0: // Idle
	IF rtWrite.Q AND NOT bBusy THEN
		bBusy 					:= TRUE;
		bError 					:= FALSE;
		udiErrorID				:= 0;
		// MinMon 16#0000_000B;	// 2B
		wSetMinMon.0 			:= bSetMinMon;
		fbADSWRITE.WRITE		:= TRUE;
		fbADSWRITE.IDXOFFS		:= 16#0000_000B;
		fbADSWRITE.LEN			:= 2;
		fbADSWRITE.SRCADDR		:= ADR(wSetMinMon);
		iStepWrite				:= iStepWrite + 5;
	END_IF
	
5, 15, 25: // Wait CMD for end
	fbADSWRITE.WRITE			:= FALSE;
	IF NOT fbADSWRITE.BUSY AND NOT fbADSWRITE.ERR THEN
		iStepWrite				:= iStepWrite + 5;
	ELSIF fbADSWRITE.ERR THEN
		iStepWrite				:= 1000;
	END_IF
	
10: // udiIDXOFFS_MinPos		: UDINT := 16#0000_000D;	// 8B
	fbADSWRITE.WRITE			:= TRUE;
	fbADSWRITE.IDXOFFS			:= 16#0000_000D;
	fbADSWRITE.LEN				:= 8;
	fbADSWRITE.SRCADDR			:= ADR(lrSetMinPos);
	iStepWrite					:= iStepWrite + 5;

20: // 	udiIDXOFFS_MaxMon		: UDINT := 16#0000_000C;	// 2B
	wSetMaxMon.0 				:= bSetMaxMon;
	fbADSWRITE.WRITE			:= TRUE;
	fbADSWRITE.IDXOFFS			:= 16#0000_000C;
	fbADSWRITE.LEN				:= 2;
	fbADSWRITE.SRCADDR			:= ADR(wSetMaxMon);
	iStepWrite					:= iStepWrite + 5;

30: // 		udiIDXOFFS_MaxPos		: UDINT := 16#0000_000E;	// 8B
	fbADSWRITE.WRITE			:= TRUE;
	fbADSWRITE.IDXOFFS			:= 16#0000_000E;
	fbADSWRITE.LEN				:= 8;
	fbADSWRITE.SRCADDR			:= ADR(lrSetMaxPos);
	iStepWrite					:= iStepWrite + 5;
		
35: // 	End
	fbADSWRITE.WRITE			:= FALSE;
	IF NOT fbADSWRITE.BUSY AND NOT fbADSWRITE.ERR THEN
		bBusy 					:= FALSE;
		iStepWrite				:= 0;
	ELSIF fbADSWRITE.ERR THEN
		iStepWrite				:= 1000;
	END_IF
	
1000:
	bBusy 						:= FALSE;
	bError 						:= TRUE;
	udiErrorID					:= fbADSWRITE.ERRID;
	iStepWrite					:= 0;

END_CASE
END_ACTION

END_FUNCTION_BLOCK

// ---- POUs/FB/FB_AxisDiag.TcPOU
//==================================================================================================
//							Beckhoff Automation Poland
//								FB_AxisDiag
//									23.08.2016
//					Blok do diagnostyki osi
// 	v1.0 || TC v 3.1.4020.0 || - pierwsza wersja
//==================================================================================================
FUNCTION_BLOCK FB_AxisDiag
VAR_INPUT
	IPCNetID								: T_AmsNetId; 	(* AmsNetId of the IPC *)
	Timeout								: TIME := DEFAULT_ADS_TIMEOUT;
	Reset								: BOOL;
	GetDiag								: BOOL;
END_VAR
VAR_IN_OUT
	Axis	 								: AXIS_REF;
	stAX5000Diag						: ST_AX5000Diag;
END_VAR
VAR_OUTPUT
	Error								: BOOL;
	AdsErrId							: UINT;
	SercosErrId							: UINT;
	ResetAct							: BOOL;
	DiagAct								: BOOL;
	Busy								: BOOL;
END_VAR
VAR
	iState								: INT;
	iSubState							: INT;
	GetDriveRef							: BOOL := TRUE;
	DriveRef								: ST_DriveRef; (* contains sNetID of EcMaster, nSlaveAddr of EcDrive, nDriveNo of EcDrive, either preset or read from NC *)
	AxisID								: UDINT;

	C1DErrorPrev							: BOOL;
	WcStateErrorPrev						: BOOL;
	AxisErrorPrev							: BOOL;
	OperationalPrev						: BOOL;
	ResetPrev							: BOOL;
	GetDiagPrev							: BOOL;

	fbSoERead							: FB_SoERead;
	fbDiagMessage 						: FB_SoEReadDiagMessage;
	fbClassXDiag							: FB_SoEReadClassXDiag;
	fbDiagNumber						: FB_SoEReadDiagNumber;
	fbDiagNumberList						: FB_SoEReadDiagNumberList;

	fbReset								: FB_SoEReset;
	fbDelay								: TON;
	fbGetSlaveState 						: FB_EcGetSlaveState;
	fbReqSlaveState 						: FB_EcReqSlaveState;
	fbNcReset 							: MC_Reset;

	fbAdsRead							: ADSREAD;
	readBuffer							: ARRAY[0..9] OF BYTE;
	Ids									: T_AmsNetIdArr;

	fbFormatString						: FB_FormatString;
	DiagMsgPrev							: STRING(255);
	LogMsg								: STRING(255);
	strSoEString							: ST_SoE_String;
	I									: INT;
END_VAR
VAR CONSTANT
	NCIDXG_AXPARMS					: UDINT := 16#00004000;	(* Axis with ID: Parameter 			*)
	NCIDXO_AXP_HWAMSADDR			: UDINT := 16#00000031;
END_VAR

stAX5000Diag.bOperational	:= Axis.NcToPlc.StateDWord.0;
stAX5000Diag.bC1DError	 	:= Axis.NcToPlc.StateDWord.28;
stAX5000Diag.bWcStateError 	:= Axis.NcToPlc.StateDWord.30;
stAX5000Diag.bAxisError		:= Axis.NcToPlc.StateDWord.31;
stAX5000Diag.iAxisErrorCode	:= Axis.NcToPlc.ErrorCode;

CASE iState OF
0:	(* idle *)
	GetDriveRef 	:= (DriveRef.nSlaveAddr = 0);

	IF GetDriveRef THEN
		Busy			:= TRUE;
		Error			:= FALSE;
		AdsErrId		:= 0;
		SercosErrId		:= 0;
		iState 			:= 1;
		iSubState		:= 0;
		AxisID 			:= Axis.NcToPlc.AxisId;

	ELSIF Reset AND NOT ResetPrev THEN
		Busy			:= TRUE;
		ResetAct		:= TRUE;
		ResetPrev		:= Reset;
		Error			:= FALSE;
		AdsErrId		:= 0;
		SercosErrId		:= 0;
		iState 			:= 2;
		iSubState		:= 0;
		AxisID 			:= Axis.NcToPlc.AxisId;

	ELSIF GetDiag AND NOT GetDiagPrev OR
		(stAX5000Diag.bC1DError AND NOT C1DErrorPrev) OR (NOT stAX5000Diag.bC1DError AND C1DErrorPrev) (* rising/falling C1D *) OR
		(stAX5000Diag.bWcStateError AND NOT WcStateErrorPrev) OR (NOT stAX5000Diag.bWcStateError AND WcStateErrorPrev) (* rising/falling WcState *) OR
		(stAX5000Diag.bAxisError AND NOT AxisErrorPrev) OR (NOT stAX5000Diag.bAxisError AND AxisErrorPrev) (* rising/falling NcError *) OR
		(stAX5000Diag.bOperational AND NOT OperationalPrev) OR (NOT stAX5000Diag.bOperational AND OperationalPrev) (* rising/falling Enable *) THEN

		Busy			:= TRUE;
		DiagAct			:= TRUE;
		GetDiagPrev		:= GetDiag;
		Error			:= FALSE;
		AdsErrId		:= 0;
		SercosErrId		:= 0;
		iState 			:= 3;
		iSubState		:= 0;
		AxisID 			:= Axis.NcToPlc.AxisId;

		(* set/clear flags *)
		C1DErrorPrev		:= stAX5000Diag.bC1DError;
		WcStateErrorPrev	:= stAX5000Diag.bWcStateError;
		AxisErrorPrev		:= stAX5000Diag.bAxisError;
		OperationalPrev		:= stAX5000Diag.bOperational;

	ELSE
		ResetAct	:= FALSE;
		DiagAct		:= FALSE;
	END_IF

1:	(* get drive reference *)
	M_GetDriveRef();

2:	(* reset and state change *)
	M_Reset();

3:	(* get diag data *)
	M_GetDiagnosis();

END_CASE

(* clear latch *)
ResetPrev	:= ResetPrev AND Reset;
GetDiagPrev	:= GetDiagPrev AND GetDiag;

ACTION M_GetDiagnosis:
CASE iSubState OF
0:	fbClassXDiag(
		NetId		:= IPCNetID,
		Execute		:= TRUE,
		DiagClass 	:= 1,
		Timeout		:= DEFAULT_ADS_TIMEOUT,
		Axis		:= Axis,
	);

	IF NOT fbClassXDiag.Busy THEN
		fbClassXDiag(Execute:= FALSE,Axis := Axis);

		IF NOT fbClassXDiag.Error THEN
			stAX5000Diag.wClass1Diag	:= fbClassXDiag.ClassXDiag;
			stAX5000Diag.stClass1Diag	:= F_ConvWordToSTAX5000C1D(stAX5000Diag.wClass1Diag);
		ELSE
			Error			:= TRUE;
			AdsErrId		:= fbClassXDiag.AdsErrId;
			SercosErrId	:= fbClassXDiag.SercosErrId;
		END_IF
		iSubState	:= iSubState + 1;
	END_IF

1:	fbDiagMessage(
		NetId	:= IPCNetID,
		Execute	:= TRUE,
		Timeout	:= DEFAULT_ADS_TIMEOUT,
		Axis	:= Axis,
	);

	IF NOT fbDiagMessage.Busy THEN
		fbDiagMessage(Execute:= FALSE,Axis := Axis);

		IF NOT fbDiagMessage.Error THEN
			stAX5000Diag.strDiagMessage := LEFT(fbDiagMessage.DiagMessage.strData, UINT_TO_INT(fbDiagMessage.DiagMessage.iActualSize));
		ELSE
			Error			:= TRUE;
			AdsErrId		:= fbDiagMessage.AdsErrId;
			SercosErrId	:= fbDiagMessage.SercosErrId;
		END_IF
		iSubState	:= iSubState + 1;
	END_IF

2:	fbDiagNumber(
		NetId	:= IPCNetID,
		Execute	:= TRUE,
		Timeout	:= DEFAULT_ADS_TIMEOUT,
		Axis	:= Axis,
	);

	IF NOT fbDiagNumber.Busy THEN
		fbDiagNumber(Execute:= FALSE,Axis := Axis);

		IF NOT fbDiagNumber.Error THEN
			stAX5000Diag.iDiagNumber := fbDiagNumber.DiagNumber;
		ELSE
			Error			:= TRUE;
			AdsErrId		:= fbDiagNumber.AdsErrId;
			SercosErrId	:= fbDiagNumber.SercosErrId;
		END_IF
		iSubState	:= iSubState + 1;
	END_IF

3:	fbSoERead(
		NetId	:= IPCNetID,
		Execute	:= TRUE,
		Idn		:= 135,
		Element	:=16#44,
		pDstBuf	:=ADR(stAX5000Diag.wDriveStatus),
		BufLen	:=SIZEOF(stAX5000Diag.wDriveStatus),
		Timeout	:= DEFAULT_ADS_TIMEOUT,
		Axis	:= Axis,
	);

	IF NOT fbSoERead.Busy THEN
		fbSoERead(Execute:= FALSE,Axis := Axis);
		IF NOT fbSoERead.Error THEN
			stAX5000Diag.stDriveStatus := F_ConvWordToSTAX5000DriveStatus(stAX5000Diag.wDriveStatus);
			iSubState		:= iSubState + 1;
		ELSE
			Error			:= TRUE;
			AdsErrId		:= fbSoERead.AdsErrId;
			SercosErrId	:= fbSoERead.SercosErrId;
			iSubState		:= iSubState + 2;
		END_IF
	END_IF

4:	fbSoERead(
		NetId	:= IPCNetID,
		Execute	:= TRUE,
		Idn		:= stAX5000Diag.stDriveStatus.iActOpModeParNum,
		Element	:=16#44,
		pDstBuf	:=ADR(stAX5000Diag.stDriveStatus.eActOpMode),
		BufLen	:=SIZEOF(stAX5000Diag.stDriveStatus.eActOpMode),
		Timeout	:= DEFAULT_ADS_TIMEOUT,
		Axis	:= Axis,
	);

	IF NOT fbSoERead.Busy THEN
		fbSoERead(Execute:= FALSE,Axis := Axis);
		IF NOT fbSoERead.Error THEN
			;
		ELSE
			Error			:= TRUE;
			AdsErrId		:= fbSoERead.AdsErrId;
			SercosErrId	:= fbSoERead.SercosErrId;
		END_IF
		iSubState	:= iSubState + 1;
	END_IF

5:	fbGetSlaveState(
		sNetId		:= DriveRef.sNetId,
		nSlaveAddr	:= DriveRef.nSlaveAddr,
		bExecute	:= TRUE,
		tTimeout	:= DEFAULT_ADS_TIMEOUT,
	);

	IF NOT fbGetSlaveState.bBusy THEN
		fbGetSlaveState(bExecute:= FALSE);
		IF NOT fbGetSlaveState.bError THEN
			stAX5000Diag.stEcSlaveState := fbGetSlaveState.state;
			stAX5000Diag.stEcSlaveStateBits := F_ConvSlaveStateToBits(fbGetSlaveState.state);
		ELSE
			Error			:= TRUE;
			AdsErrId		:= UDINT_TO_UINT(fbGetSlaveState.nErrId);
		END_IF

		IF stAX5000Diag.stEcSlaveStateBits.bError THEN
			IF stAX5000Diag.stEcSlaveStateBits.bPreop THEN
				(* read S21 - IDN List of Invalid operation data for CP2 (Preop->SaveOp) *)
				MEMSET(ADR(stAX5000Diag.stCPxInvParamList), 0, SIZEOF(stAX5000Diag.stCPxInvParamList));
				stAX5000Diag.bPreopToSafeOpError := TRUE;
				stAX5000Diag.bSafeOpToOpError := FALSE;
				iSubState	:= iSubState + 1;
			ELSIF stAX5000Diag.stEcSlaveStateBits.bSafeOp THEN
				(* read S22 - IDN List of Invalid operation data for CP3 (SaveOp->Op) *)
				MEMSET(ADR(stAX5000Diag.stCPxInvParamList), 0, SIZEOF(stAX5000Diag.stCPxInvParamList));
				stAX5000Diag.bPreopToSafeOpError := FALSE;
				stAX5000Diag.bSafeOpToOpError := TRUE;
				iSubState	:= iSubState + 2;
			ELSE
				(* Skip S21 + S22 *)
				MEMSET(ADR(stAX5000Diag.stCPxInvParamList), 0, SIZEOF(stAX5000Diag.stCPxInvParamList));
				stAX5000Diag.bPreopToSafeOpError := FALSE;
				stAX5000Diag.bSafeOpToOpError := FALSE;
				iSubState	:= iSubState + 3;
			END_IF
		ELSE
			(* Skip S21 + S22 *)
			MEMSET(ADR(stAX5000Diag.stCPxInvParamList), 0, SIZEOF(stAX5000Diag.stCPxInvParamList));
			stAX5000Diag.bPreopToSafeOpError := FALSE;
			stAX5000Diag.bSafeOpToOpError := FALSE;
			iSubState	:= iSubState + 3;
		END_IF
	END_IF

6:	(* read S21 - IDN List of Invalid operation data for CP2 (Preop->SaveOp) *)
	fbSoERead(
		NetId	:= IPCNetID,
		Execute	:= TRUE,
		Idn		:= 21,
		Element	:=16#40,
		pDstBuf	:=ADR(stAX5000Diag.stCPxInvParamList),
		BufLen	:=SIZEOF(stAX5000Diag.stCPxInvParamList),
		Timeout	:= DEFAULT_ADS_TIMEOUT,
		Axis	:= Axis,
	);

	IF NOT fbSoERead.Busy THEN
		fbSoERead(Execute:= FALSE,Axis := Axis);
		IF NOT fbSoERead.Error THEN
			;
		ELSE
			Error			:= TRUE;
			AdsErrId		:= fbSoERead.AdsErrId;
			SercosErrId	:= fbSoERead.SercosErrId;
		END_IF
		iSubState	:= iSubState + 2;
	END_IF

7:	(* read S22 - IDN List of Invalid operation data for CP3 (SaveOp->Op) *)
	fbSoERead(
		NetId	:= IPCNetID,
		Execute	:= TRUE,
		Idn		:= 22,
		Element	:=16#40,
		pDstBuf	:=ADR(stAX5000Diag.stCPxInvParamList),
		BufLen	:=SIZEOF(stAX5000Diag.stCPxInvParamList),
		Timeout	:= DEFAULT_ADS_TIMEOUT,
		Axis	:= Axis,
	);

	IF NOT fbSoERead.Busy THEN
		fbSoERead(Execute:= FALSE,Axis := Axis);
		IF NOT fbSoERead.Error THEN
			;
		ELSE
			Error			:= TRUE;
			AdsErrId		:= fbSoERead.AdsErrId;
			SercosErrId	:= fbSoERead.SercosErrId;
		END_IF
		iSubState	:= iSubState + 1;
	END_IF

8:	fbDiagNumberList(
		NetId			:= IPCNetID,
		Execute			:= TRUE,
		Timeout			:= DEFAULT_ADS_TIMEOUT,
		pDiagNumber		:= ADR(stAX5000Diag.stDiagNumberList),
		Size			:= SIZEOF(stAX5000Diag.stDiagNumberList),
		Axis			:= Axis,
	);

	IF NOT fbDiagNumberList.Busy THEN
		fbDiagNumberList(Execute:= FALSE,Axis := Axis);

		IF NOT fbDiagNumberList.Error THEN
			IF GVL_AXIS.bLogDriveDiagMsgs THEN
				IF (stAX5000Diag.strDiagMessage <> DiagMsgPrev) AND (stAX5000Diag.stDiagNumberList.iActualSize > 0) THEN

					fbFormatString(
						sFormat := 'Axis ID: %d, DriveDiag: ',
						arg1 := F_UDINT(AxisID),
						sOut => LogMsg
					);
	
					FOR I := 0 TO MIN(29, UINT_TO_INT(stAX5000Diag.stDiagNumberList.iActualSize)/4-1) DO
						IF (stAX5000Diag.stDiagNumberList.arrDiagNumbers[I] <> 0) THEN
							fbFormatString(
								sFormat := '%X, ',
								arg1 := F_UDINT(stAX5000Diag.stDiagNumberList.arrDiagNumbers[I])
							);
	
							LogMsg := CONCAT(LogMsg, fbFormatString.sOut);
						END_IF
					END_FOR
	
					LogMsg := CONCAT(LogMsg, 'DiagMsg: ');
					LogMsg := CONCAT(LogMsg, stAX5000Diag.strDiagMessage);
	
					(* report message *)
					ADSLOGSTR(msgCtrlMask := ADSLOG_MSGTYPE_ERROR OR ADSLOG_MSGTYPE_LOG,
						msgFmtStr := LogMsg, strArg:= '');
	
					DiagMsgPrev := stAX5000Diag.strDiagMessage;
				END_IF
			END_IF
		ELSE
			Error			:= TRUE;
			AdsErrId		:= fbDiagNumberList.AdsErrId;
			SercosErrId	:= fbDiagNumberList.SercosErrId;
		END_IF

		IF (stAX5000Diag.strMotorType = '') OR (stAX5000Diag.strDriveType = '') THEN
			iSubState	:= iSubState + 1;
		ELSE
			DiagAct	:= FALSE;
			iSubState	:= 0;
			iState		:= 0;
			Busy		:= FALSE;
		END_IF
	END_IF

9:	fbSoERead(
		NetId	:= IPCNetID,
		Execute	:= TRUE,
		Idn		:= P_0_IDN + 53,
		Element	:=16#44,
		pDstBuf	:=ADR(strSoEString),
		BufLen	:=SIZEOF(strSoEString),
		Timeout	:= DEFAULT_ADS_TIMEOUT,
		Axis	:= Axis,
	);

	IF NOT fbSoERead.Busy THEN
		fbSoERead(Execute:= FALSE,Axis := Axis);
		IF NOT fbSoERead.Error THEN
			MEMSET(ADR(stAX5000Diag.strMotorType),0,SIZEOF(stAX5000Diag.strMotorType));
			MEMCPY(ADR(stAX5000Diag.strMotorType),ADR(strSoEString.strData),MIN(SIZEOF(stAX5000Diag.strMotorType),strSoEString.iActualSize));
		ELSE
			Error			:= TRUE;
			AdsErrId		:= fbSoERead.AdsErrId;
			SercosErrId	:= fbSoERead.SercosErrId;
		END_IF
		iSubState	:= iSubState + 1;
	END_IF

10:	fbSoERead(
		NetId	:= IPCNetID,
		Execute	:= TRUE,
		Idn		:= P_0_IDN + 324,
		Element	:=16#44,
		pDstBuf	:=ADR(strSoEString),
		BufLen	:=SIZEOF(strSoEString),
		Timeout	:= DEFAULT_ADS_TIMEOUT,
		Axis	:= Axis,
	);

	IF NOT fbSoERead.Busy THEN
		fbSoERead(Execute:= FALSE,Axis := Axis);
		IF NOT fbSoERead.Error THEN
			MEMSET(ADR(stAX5000Diag.strDriveType),0,SIZEOF(stAX5000Diag.strDriveType));
			MEMCPY(ADR(stAX5000Diag.strDriveType),ADR(strSoEString.strData),MIN(SIZEOF(stAX5000Diag.strDriveType),strSoEString.iActualSize));
		ELSE
			Error			:= TRUE;
			AdsErrId		:= fbSoERead.AdsErrId;
			SercosErrId	:= fbSoERead.SercosErrId;
		END_IF
		DiagAct	:= FALSE;
		iSubState	:= 0;
		iState		:= 0;
		Busy		:= FALSE;
	END_IF


END_CASE
END_ACTION

ACTION M_GetDriveRef:
(* get reference from NC *)
fbAdsRead(
	NETID	:= IPCNetID,
	PORT	:= AMSPORT_R0_NC,
	IDXGRP	:= NCIDXG_AXPARMS + Axis.NcToPlc.AxisId,
	IDXOFFS	:= NCIDXO_AXP_HWAMSADDR,
	LEN		:= SIZEOF(readBuffer) ,
	DESTADDR:= ADR(readBuffer),
	READ	:= TRUE,
	TMOUT	:= Timeout
);

IF NOT fbAdsRead.BUSY THEN
	fbAdsRead(READ := FALSE);
	stAX5000Diag.nNCAxisID := Axis.NcToPlc.AxisId;

	IF NOT fbAdsRead.ERR THEN
		MEMCPY(ADR(Ids), ADR(readBuffer), SIZEOF(Ids)); 										(* readBuffer[0..5] *)
		MEMCPY(ADR(DriveRef.nSlaveAddr), ADR(readBuffer[6]), SIZEOF(DriveRef.nSlaveAddr));  	(* readBuffer[6..7] *)
		MEMCPY(ADR(DriveRef.nDriveNo), ADR(readBuffer[8]), SIZEOF(DriveRef.nDriveNo));  		(* readBuffer[8..9] *)

		(* create string out of byte array *)
		DriveRef.sNetId := F_CreateAmsNetId(Ids);
		GetDriveRef := FALSE;
	END_IF

	Busy	:= FALSE;
	iState	:= 0;
END_IF
END_ACTION

ACTION M_Reset:
CASE iSubState OF
0:
	IF stAX5000Diag.bWcStateError OR stAX5000Diag.bC1DError THEN
		(* ResetAmplifier *)
		iSubState := iSubState + 1;
	ELSIF stAX5000Diag.stEcSlaveStateBits.bError AND GVL_Axis.bForceStateChgAfterDrvReset THEN
		(* Clear Error *)
		iSubState := 4;
	ELSIF (NOT stAX5000Diag.bOperational) OR stAX5000Diag.bAxisError OR (stAX5000Diag.iAxisErrorCode <> 0) THEN
		(* NC Reset only *)
		iSubState := 6;
	ELSE
		(* reset not required *)
		iSubState	:= 0;
		iState		:= 0;
		Busy		:= FALSE;
		ResetAct	:= FALSE;
	END_IF

1:	(* ResetAmplifier *)
	fbReset(
		NetId	:= IPCNetID,
		Execute	:= TRUE,
		Timeout	:= DEFAULT_ADS_TIMEOUT,
		Axis	:= Axis,
	);
	IF NOT fbReset.Busy THEN
		fbReset(Execute:= FALSE, Axis:= Axis);

		IF NOT fbReset.Error THEN
			IF GVL_Axis.bLogDriveDiagMsgs THEN
				LogMsg := CONCAT('Axis ID: ', DWORD_TO_STRING(Axis.NcToPlc.AxisId));
				LogMsg := CONCAT(LogMsg, ', Drive Reset');

				(* report message *)
				ADSLOGSTR(msgCtrlMask := ADSLOG_MSGTYPE_ERROR OR ADSLOG_MSGTYPE_LOG,
					msgFmtStr := LogMsg, strArg:= '');

				DiagMsgPrev := '';
			END_IF
			iSubState	:= iSubState + 1;
		ELSE
			Error			:= TRUE;
			AdsErrId		:= fbReset.AdsErrId;
			SercosErrId	:= fbReset.SercosErrId;
			Busy			:= FALSE;
			ResetAct		:= FALSE;
			iSubState		:= 0;
			iState			:= 0;
		END_IF
	END_IF

2:	fbDelay(IN:=TRUE, PT:=t#3s);
	IF fbDelay.Q THEN
		fbDelay(IN:=FALSE);
		iSubState	:= iSubState + 1;
	END_IF

3:	fbGetSlaveState(
		sNetId		:= DriveRef.sNetId,
		nSlaveAddr	:= DriveRef.nSlaveAddr,
		bExecute	:= TRUE,
		tTimeout	:= DEFAULT_ADS_TIMEOUT,
	);

	IF NOT fbGetSlaveState.bBusy THEN
		fbGetSlaveState(bExecute:= FALSE);

		IF NOT fbGetSlaveState.bError THEN
			IF ((fbGetSlaveState.state.deviceState <> 16#08) OR ((fbGetSlaveState.state.deviceState AND 16#10) = 16#10)) AND
				GVL_Axis.bForceStateChgAfterDrvReset THEN

				iSubState	:= iSubState + 1;
			ELSIF Axis.NcToPlc.StateDWord.31 OR (Axis.NcToPlc.ErrorCode <> 0) THEN
				iSubState	:= 6;
			ELSE
				Busy		:= FALSE;
				ResetAct	:= FALSE;
				iSubState	:= 0;
				iState		:= 0;
			END_IF
		ELSE
			Error			:= TRUE;
			AdsErrId		:= UDINT_TO_UINT(fbGetSlaveState.nErrId);
			Busy			:= FALSE;
			ResetAct		:= FALSE;
			iSubState		:= 0;
			iState			:= 0;
		END_IF
	END_IF

4:	(* clear error *)
	fbReqSlaveState(
		sNetId		:= DriveRef.sNetId,
		nSlaveAddr	:= DriveRef.nSlaveAddr,
		bExecute	:= TRUE,
		tTimeout	:= DEFAULT_ADS_TIMEOUT,
		state		:= EC_DEVICE_STATE_ERROR);

	IF NOT fbReqSlaveState.bBusy THEN
		fbReqSlaveState(bExecute:= FALSE);

		IF NOT fbReqSlaveState.bError THEN
			iSubState	:= iSubState + 1;
		ELSE
			Error		:= TRUE;
			AdsErrId	:= UDINT_TO_UINT(fbReqSlaveState.nErrId);
			Busy		:= FALSE;
			ResetAct	:= FALSE;
			iSubState	:= 0;
			iState		:= 0;
		END_IF
	END_IF

5:	(* set op *)
	fbReqSlaveState(
		sNetId		:= DriveRef.sNetId,
		nSlaveAddr	:= DriveRef.nSlaveAddr,
		bExecute	:= TRUE,
		tTimeout	:= DEFAULT_ADS_TIMEOUT,
		state		:= EC_DEVICE_STATE_OP);

	IF NOT fbReqSlaveState.bBusy THEN
		fbReqSlaveState(bExecute:= FALSE);

		IF NOT fbReqSlaveState.bError THEN
			iSubState	:= iSubState + 1;
		ELSE
			Error		:= TRUE;
			AdsErrId	:= UDINT_TO_UINT(fbReqSlaveState.nErrId);
			Busy		:= FALSE;
			ResetAct	:= FALSE;
			iSubState	:= 0;
			iState		:= 0;
		END_IF
	END_IF

6:	fbNcReset(
		Execute:= TRUE,
		Axis:= Axis,
	);
	IF fbNcReset.Done OR fbNcReset.Error THEN
		IF fbNcReset.Error THEN
			Error 		:= TRUE;
			AdsErrId 	:= UDINT_TO_UINT(fbNcReset.ErrorID);
		END_IF

		iSubState	:= 0;
		iState		:= 0;
		Busy		:= FALSE;
		ResetAct	:= FALSE;
		fbNcReset(Execute:= FALSE, Axis:= Axis);
	END_IF
END_CASE
END_ACTION

END_FUNCTION_BLOCK

// ---- POUs/Programy/Hbot/AxisOnline/POUsAxisOnline/FBs/FB_GetDriveRef.TcPOU
//==================================================================================================
//							Beckhoff Automation Poland
//									28.03.2018
//	Blok funkcyjny tworzacy strukture ST_DriveRef z AXIS_REF
//	Przydatny w komunikacji CoE w AX8000
//  v1.0	|| TC v 3.1.4022.16		|| - pierwsza wersja
//==================================================================================================
FUNCTION_BLOCK FB_GetDriveRef
VAR_INPUT
	bExecute								: BOOL;							// rising edge starts sequence
END_VAR
VAR_OUTPUT
	bBusy									: BOOL;
	bError									: BOOL;	
	udiErrorID								: UDINT;						// bError=TRUE AND udiErrorID=0 means state request timeout
	stDriveRef								: ST_DriveRef;					// come from stPlcDriveRef
END_VAR
VAR_IN_OUT
	Axis									: AXIS_REF;
END_VAR
VAR
	fbAdsRead								: ADSREAD;
	ftADSRead								: F_TRIG;
	stPlcDriveRef							: ST_PlcDriveRef;				// ADS buffer (need to change aNetId into sNetId)
END_VAR
VAR CONSTANT
	NCIDXG_AXPARMS							: UDINT			:= 16#4000;		// ADS group number to axis parameters 
	NCIDXO_AXP_HWAMSADDR					: UDINT			:= 16#31;		// ADS offset to drive channel
END_VAR

fbAdsRead(	NETID			:= '', 
			PORT			:= AMSPORT_R0_NC, 								// set ADS Port to NC
			IDXGRP			:= NCIDXG_AXPARMS + Axis.NcToPlc.AxisId,		// set ADS Group to AXIS Parameters 
			IDXOFFS			:= NCIDXO_AXP_HWAMSADDR,						// set ADS offset to channel number 
			LEN				:= SIZEOF(stPlcDriveRef), 
			DESTADDR		:= ADR(stPlcDriveRef), 
			READ			:= bExecute, 
			BUSY			=> bBusy, 
			ERR				=> bError, 
			ERRID			=> udiErrorID);
			
ftADSRead(CLK:= bBusy);

IF ftADSRead.Q AND NOT fbAdsRead.ERR THEN	
	stDriveRef.sNetId		:= F_CreateAmsNetId(stPlcDriveRef.aNetId);		// change AmsNetId array into string
	stDriveRef.nSlaveAddr	:= stPlcDriveRef.nSlaveAddr;
	stDriveRef.nDriveNo		:= stPlcDriveRef.nDriveNo;			
END_IF

END_FUNCTION_BLOCK

// ---- POUs/FB/FB_MX2.TcPOU
FUNCTION_BLOCK FB_MX2
VAR_INPUT
	b_CW   AT%I*  :BOOL;
	b_CCW AT%I*  :BOOL;
	b_Reset AT%I* :BOOL;
	ui_CzestotliwoscI AT %I*: INT;
	w_Status AT%I* :WORD;
	udi_RampaACC_in AT %I*: WORD;
	udi_RampaDCC_in AT %I*: WORD;
END_VAR
	
	
VAR_OUTPUT
	ui_CzestotliwoscO AT %Q*: INT;
	udi_RampaACC_out AT %Q*: WORD;
	udi_RampaDCC_out AT %Q*: WORD;
	b_Rady AT %Q*: BOOL;
	b_Pracuje AT %Q*: BOOL;
	w_ControlW AT%Q* :WORD;
	Blad AT%Q* :BOOL;
END_VAR

VAR
	
	LokRem : BOOL;
	DoPrzodu :BOOL;
	DoTylu:BOOL;
	BladFalownik :BOOL;
	BladFalownikKom :BOOL;
	out1 :WORD;
	out2 :WORD;
	out3 :WORD;
	out4 :WORD;
	out5 :WORD;
	OP_O :TON;
	axal_Fal : BOOL;
	OP_50Hax : TON;
	OP_Hax :TON;
	Fal_s :INT;
	OP_Falownik_OFF :TON;
	Wyl_Fal :BOOL;
	
	
	
	Wylacz: BOOL;
END_VAR

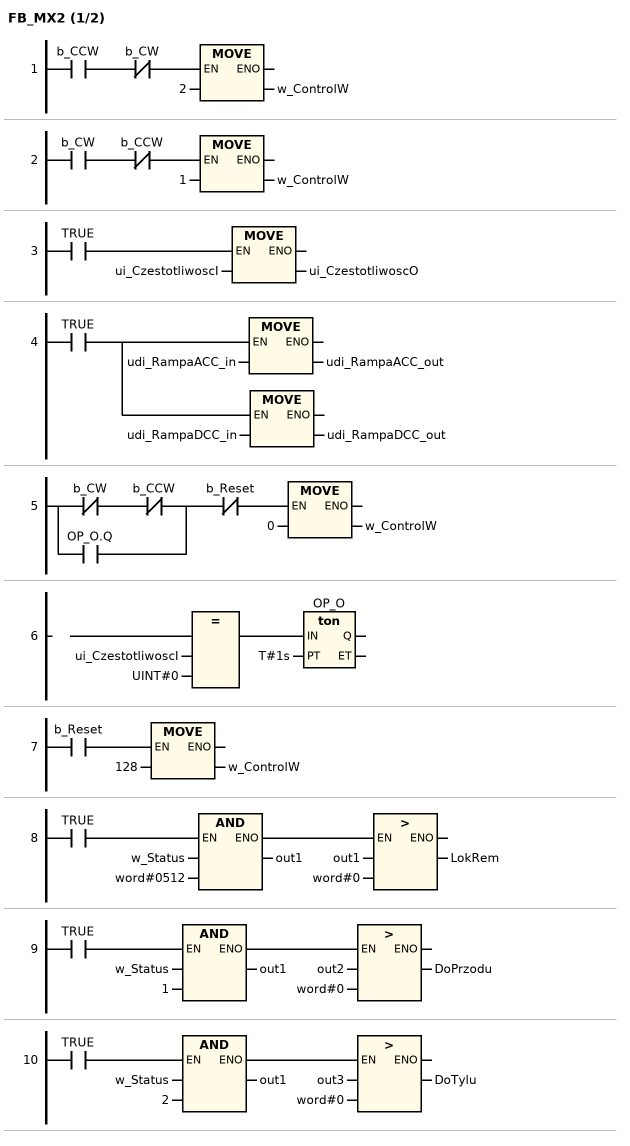
// NETWORK 1
IF b_CCW AND NOT b_CW THEN w_ControlW := 2; END_IF

// NETWORK 2
IF b_CW AND NOT b_CCW THEN w_ControlW := 1; END_IF

// NETWORK 3
ui_CzestotliwoscO := ui_CzestotliwoscI;

// NETWORK 4
udi_RampaACC_out := udi_RampaACC_in;
udi_RampaDCC_out := udi_RampaDCC_in;

// NETWORK 5
IF (NOT b_CW AND NOT b_CCW OR OP_O.Q) AND NOT b_Reset THEN w_ControlW := 0; END_IF

// NETWORK 6
OP_O(IN := ui_CzestotliwoscI = UINT#0, PT := T#1s); // ton

// NETWORK 7
IF b_Reset THEN w_ControlW := 128; END_IF

// NETWORK 8
out1 := w_Status AND word#0512;
LokRem := out1 > word#0;

// NETWORK 9
out1 := w_Status AND 1;
DoPrzodu := out2 > word#0;

// NETWORK 10
out1 := w_Status AND 2;
DoTylu := out3 > word#0;

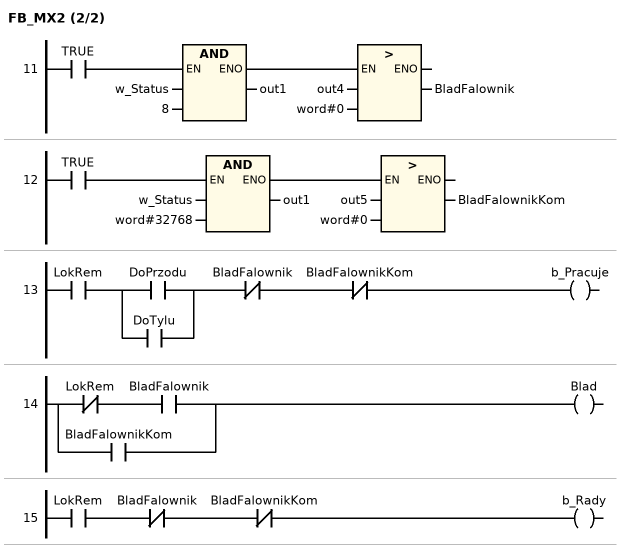
// NETWORK 11
out1 := w_Status AND 8;
BladFalownik := out4 > word#0;

// NETWORK 12
out1 := w_Status AND word#32768;
BladFalownikKom := out5 > word#0;

// NETWORK 13
b_Pracuje := LokRem AND (DoPrzodu OR DoTylu) AND NOT BladFalownik AND NOT BladFalownikKom;

// NETWORK 14
Blad := NOT LokRem AND BladFalownik OR BladFalownikKom;

// NETWORK 15
b_Rady := LokRem AND NOT BladFalownik AND NOT BladFalownikKom;

END_FUNCTION_BLOCK

// ---- POUs/FB/FB_Prawidlo.TcPOU
PROGRAM FB_Prawidlo
VAR
			//internals
			
			i_seq :INT;
			Czas :ARRAY[0..100] OF TON;
			wyzwolenie         :R_TRIG;
END_VAR

VAR_INPUT			
			//in
			b_Start AT %I* :BOOL;
			b_Stop AT %I* :BOOL;
			bKon_Hamulec1 AT%I* :BOOL	; //kontraktron hamulec 1
			bKon_Hamulec2 AT%I* :BOOL	; //kontraktron hamulec 2
			bKonPodajnik1 AT%I* :BOOL	; //kontraktron podajnik 1
			bKonPodajnik2 AT%I* :BOOL	; //kontraktron podajnik 2
			bCzHamulec AT%I* :BOOL	; //czujnik hamulec 
			bZaladowany AT%I* :BOOL	; //czujnik hamulec 
END_VAR
 //OUT	
VAR_OUTPUT

			 bZaworPodnosnik1 AT%Q* :BOOL	;	// cewka podnośnik 1
			 bZaworPodnosnik2 AT%Q* :BOOL	;	// cewka podnośnik 2
			 bZaworHamulec AT%Q* :BOOL	;	// cewka hamulec
	 		 bZgodaNaRuch AT%Q* :BOOL	;	// cewka hamulec
			 bLaduj AT%Q* :BOOL	;	// czeka na ladunek 
END_VAR

CASE i_seq OF 
	
0:(*inicjalizacja i info o starcie *)


	bZaworPodnosnik1	:=TRUE;
	bZaworPodnosnik2	:=FALSE;
	bZaworHamulec		:=FALSE;
	bZgodaNaRuch 		:=FALSE;
	bLaduj				:=FALSE;
		 
		 IF b_Start=TRUE  THEN
		
		 
		 i_seq:=5;
		 
		END_IF

5:(*jeśli start to podnieś prawidlo do gory wystaw bita że można wydać pudełko  *)

		
			 bZgodaNaRuch		:=TRUE;
			 bZaworHamulec		:=TRUE;
			 
		 IF bKon_Hamulec1=TRUE THEN	 
			 i_seq:=10;
		 END_IF
		 
10:(*jeśli zgoda na ruch to czeka na czujnik  *)	 

	IF Czas[0].Q=TRUE THEN
		
		bZaworPodnosnik1	:=FALSE;
		bZaworPodnosnik2	:=TRUE;
	
		i_seq:=15;
	
	
	END_IF

15:(*czeka na załadunek *)	 

	IF bKonPodajnik1=TRUE THEN
		
	
		bLaduj				:=TRUE;
		i_seq:=20;
	END_IF

20:(*zaladowywuje *)	 

	IF wyzwolenie.Q=TRUE THEN
		bZaworPodnosnik1	:=TRUE;
		bZaworPodnosnik2	:=FALSE;
	i_seq:=25;
	
	END_IF
25:(*zwalnia hamulec i wraca do punktu wyjścia  *)

	IF czas[1].Q=TRUE THEN
	bZaworHamulec		:=FALSE;	
	bLaduj				:=FALSE;
	i_seq:=30;		
	
	END_IF
	
30:

	IF czas[2].Q=TRUE AND bCzHamulec=FALSE  THEN

	i_seq:=5;	
	
	END_IF

	
	

END_CASE

Czas[0](IN:=bCzHamulec, PT:=T#200MS);
Czas[1](IN:=i_seq=25, PT:=T#1S);
Czas[2](IN:=i_seq=30, PT:=T#2S);

		IF b_Stop=TRUE THEN
			
		i_seq:=0;
		
		END_IF
		wyzwolenie(CLK:=bZaladowany);

END_PROGRAM

// ---- POUs/Programy/Hbot/PRG_KinTrans.TcPOU
PROGRAM PRG_KinTrans
VAR_INPUT
	bBuildKinGroup					: BOOL; 
	bCleanKinGroup					: BOOL; 
	bResetKinGroup					: BOOL; 
END_VAR

VAR
	//Kinematic Tranformation Variables 
	fbKinConfigGroup				: FB_KinConfigGroup;
	fbKinResetGroup 				: FB_KinResetGroup;

	stKinAxes						: ST_KinAxes;
	in_stKinToPlc	AT %I*			: NcToPlc_NciChannel_Ref;
	out_stPlcToKin	AT %Q*			: PLCTONC_NCICHANNEL_REF;

	iKinState						: INT;		// Kinematics case Steps
	bAllAxesReady					: BOOL;
	
	rtKinGroup						: R_TRIG;	// Configuration of kinemtic trigger
	rtKinRegroup					: R_TRIG;	// Diasabling of kinemtic trigger
	rtKinReset						: R_TRIG;	// Reseting of kinemtic trigger


END_VAR

VAR_OUTPUT
	bKinBusy						: BOOL;
	bKinDone						: BOOL;
	bKinBuilt						: BOOL;		// Cartesian mode Enabled - check
	bKinClined						: BOOL;  	// Disable Cartesian -  command	
	//Errors	
	bKinError						: BOOL;		// Kinematic Configuration Error 
	udiKinErrorID					: UDINT;		// Kinematic Configuration Error 	
	eKinStatus						: E_KinStatus;(*KinStatus_Error,         
													KinStatus_Empty,         
													KinStatus_Unknown,    
													KinStatus_StartPending, 
													KinStatus_Ready,       
													KinStatus_InvalidItfVersion := 16#4000*)
END_VAR

stKinAxes.nAxisIdsMcs[1]	:= P_Hbot_V3.Axis_MCS_X.NcToPlc.AxisId;
stKinAxes.nAxisIdsMcs[2]	:= P_Hbot_V3.Axis_MCS_Y.NcToPlc.AxisId;
stKinAxes.nAxisIdsAcs[1]	:= P_Hbot_V3.Axis_ACS_X.NcToPlc.AxisId;
stKinAxes.nAxisIdsAcs[2]	:= P_Hbot_V3.Axis_ACS_Y.NcToPlc.AxisId;

bAllAxesReady:= P_Hbot_V3.stMcAxisOnline_MCS_X.stStatus.bAxisReady AND 
				P_Hbot_V3.stMcAxisOnline_MCS_Y.stStatus.bAxisReady AND 
				P_Hbot_V3.stMcAxisOnline_ACS_X.stStatus.bAxisReady AND 
				P_Hbot_V3.stMcAxisOnline_ACS_Y.stStatus.bAxisReady;


// Rising edge singnal - enabling kinematic
	rtKinGroup(CLK:= bAllAxesReady AND bBuildKinGroup);
// Rising edge singnal - disabling kinematic
	rtKinRegroup(CLK:= bCleanKinGroup);
	rtKinReset(CLK:= bResetKinGroup);
// Checking actual kinematic status
	eKinStatus := F_KinGetChnOperationState(stKinRefIn:= in_stKinToPlc);
	
CASE iKinState OF 
	0:	
		IF rtKinGroup.Q THEN
			iKinState := iKinState + 10;
		ELSIF rtKinregroup.Q  THEN
			iKinState := iKinState + 20; 
		ELSIF rtKinReset.Q  THEN
			iKinState := iKinState + 30; 
		END_IF
		
		fbKinConfigGroup(stAxesList				:= stKinAxes, 
						stKinRefIn				:= in_stKinToPlc, 
						bBusy					=> bKinBusy, 
						bDone					=> bKinDone,
						bError					=> bKinError, 
						nErrorId				=> udiKinErrorID);
		
	10:
		bKinError := FALSE;
		fbKinConfigGroup(bExecute			:= TRUE , 
					bCartesianMode			:= TRUE, 
					stAxesList				:= stKinAxes, 
					stKinRefIn				:= in_stKinToPlc, 
					bBusy					=> bKinBusy, 
					bDone					=> bKinDone,
					bError					=> bKinError, 
					nErrorId				=> udiKinErrorID);
		IF NOT fbKinConfigGroup.bBusy THEN
			IF fbKinConfigGroup.bError THEN
				iKinState := 999;
				bKinError := TRUE;
			ELSE
				bKinBuilt := TRUE;
				bKinClined							:= FALSE;
				iKinState := 0;
			END_IF
			fbKinConfigGroup(bExecute				:= FALSE , 
							stAxesList				:= stKinAxes, 
							stKinRefIn				:= in_stKinToPlc);
		END_IF
	20:
		bKinError := FALSE;
		fbKinConfigGroup(bExecute			:= TRUE , 
					bCartesianMode			:= FALSE, 
					stAxesList				:= stKinAxes, 
					stKinRefIn				:= in_stKinToPlc, 
					bBusy					=> bKinBusy, 
					bDone					=> bKinDone,
					bError					=> bKinError, 
					nErrorId				=> udiKinErrorID);
		IF NOT fbKinConfigGroup.bBusy THEN
			IF fbKinConfigGroup.bError THEN
				iKinState := 999;
				bKinError := TRUE;
			ELSE
				bKinBuilt							:= FALSE;
				bKinClined							:= TRUE;
				iKinState := 0;
			END_IF
			fbKinConfigGroup(bExecute				:= FALSE , 
				stAxesList				:= stKinAxes, 
				stKinRefIn				:= in_stKinToPlc);
		END_IF
	30:
		fbKinResetGroup(bExecute			:= TRUE , 
						nItpChannelId		:= in_stKinToPlc.ChnId, 
						stKinRefIn			:= in_stKinToPlc , 
						stAxesList			:= stKinAxes , 
						bBusy				=> bKinBusy , 
						bDone				=> bKinDone , 
						bError				=> bKinError , 
						nErrorId			=> udiKinErrorID );	
		
		IF NOT fbKinResetGroup.bBusy THEN
			IF fbKinResetGroup.bError THEN
				iKinState := 999;
				bKinError := TRUE;
			ELSE
				iKinState := 0;
			END_IF
			fbKinResetGroup(bExecute	:= FALSE , 
							nItpChannelId			:= in_stKinToPlc.ChnId, 
							stKinRefIn				:= in_stKinToPlc , 
							stAxesList				:= stKinAxes );	
		END_IF
	999:
		iKinState := 0;
END_CASE

END_PROGRAM

// ---- POUs/Programy/Hbot/NCI/PRG_ChannelHandler.TcPOU
PROGRAM PRG_ChannelHandler
VAR
nChan:uint;
	nOldSelectedChannel		: 	UDINT;
	fbNCIChannel1: 			FB_NCIChannel;	
END_VAR

(* ==========================================================*)
(*   FB: FB_ChannelHandler		                             *)
(* ----------------------------------------------------------*)
(*   Desc:  										         *)
(*   Auth: TV                                                *)
(*   Date: 02.04.2013                                        *)
(*   Last: 02.04.2013                                        *)
(*   Rev.: 1.0                                               *)
(* ==========================================================*)

// Channel 1 is PTP Channel

(****************************************************************************************)
(*	  Map CNC function selection from HMI to selected channel (and state vice versa)  	*)
(****************************************************************************************)
IF (nOldSelectedChannel <>INT_TO_UDINT(PLCSelectedChannel)) THEN
	PLCChannelSignals.SingleBlock 		:= PLCMachineMode[PLCSelectedChannel].SingleBlock;
	PLCChannelSignals.PrgBlockIgnore	:= PLCMachineMode[PLCSelectedChannel].PrgBlockIgnore;
	PLCChannelSignals.M01Stop 			:= PLCMachineMode[PLCSelectedChannel].M01Stop;
	PLCChannelSignals.Backward 			:= PLCMachineMode[PLCSelectedChannel].Backward;
	PLCChannelSignals.FeedHold 			:= PLCMachineMode[PLCSelectedChannel].FeedHold;
	nOldSelectedChannel 				:= INT_TO_UDINT(PLCSelectedChannel);
END_IF

PLCMachineMode[PLCSelectedChannel].SingleBlock 		:= PLCChannelSignals.SingleBlock;
PLCMachineMode[PLCSelectedChannel].PrgBlockIgnore 	:= PLCChannelSignals.PrgBlockIgnore;
PLCMachineMode[PLCSelectedChannel].M01Stop 			:= PLCChannelSignals.M01Stop;
PLCMachineMode[PLCSelectedChannel].Backward 		:= PLCChannelSignals.Backward;
PLCMachineMode[PLCSelectedChannel].FeedHold 		:= PLCChannelSignals.FeedHold;
//PLCMachineMode[PLCSelectedChannel].Reset 			:= PLCReset;

// First NC I Channel, default Channel ID=2 
nChan:=GVL_NCI.nChan;

fbNCIChannel1(
	nChan:=nChan ,

	(* Operation Mode *)
	bModeStandby := 			PLCMachineMode[nChan].Standby,
	bModeAutomatic :=			PLCMachineMode[nChan].Automatic,
	bModeManual :=				PLCMachineMode[nChan].Manual,
	bModeMDI :=					PLCMachineMode[nChan].MDI,
	bModeReference :=			PLCMachineMode[nChan].Homing,

	(* Operation State *)
	bStateStart:= 				PLCMachineMode[nChan].Start,
	bStateStop:= 				PLCMachineMode[nChan].Stop,
	bStateReset:= 				PLCMachineMode[nChan].Reset,
	(*Error*)
	bStateError:=				PLCMachineMode[nChan].Error,
	(* Special Functions *)
	bBackwardMotion:= 			PLCMachineMode[nChan].Backward,
	bPrgBlockIgnore:= 			PLCMachineMode[nChan].PrgBlockIgnore,
	bFeedHold:= 				PLCMachineMode[nChan].FeedHold,
	bSingleBlock:= 				PLCMachineMode[nChan].SingleBlock,
	bDoSingleBlock:= 			PLCMachineMode[nChan].DoSingleBlock,

	(* Strings *)
	sProgramName := 			PLCMachineMode[nChan].ProgramName,
	sMDIString :=				PLCMachineMode[nChan].MDIString );

END_PROGRAM

// ---- POUs/Programy/Hbot/NCI/2_GROUPS/FB_NCIChannel.TcPOU
FUNCTION_BLOCK FB_NCIChannel
VAR_INPUT
	nChan: 						UINT;
END_VAR

VAR_IN_OUT
	(* Operation Mode *)
	bModeStandby:				BOOL;
	bModeAutomatic:				BOOL;
	bModeManual:				BOOL;
	bModeMDI:					BOOL;
	bModeReference:				BOOL;

	(* Special Functions *)
	bBackwardMotion:			BOOL;
	bPrgBlockIgnore:			BOOL;
	bFeedHold:					BOOL;
	bSingleBlock:				BOOL;
	bDoSingleBlock:				BOOL;

	(* Operation State *)
	bStateStop:					BOOL;
	bStateReset:				BOOL;
	bStateStart: 				BOOL;
	bStateError:				BOOL; (*PiotrB*)

	(* Strings *)
	sProgramName	: 			STRING(1024);
	sMDIString		: 			STRING(1024);
END_VAR

VAR
	ItpReset1: 					ItpResetEx2;	
	fbRTrigAuto: 				R_TRIG;
	fbRTrigManual: 				R_TRIG;
	fbRTrigMDI: 				R_TRIG;
	fbRTrigReference: 			R_TRIG;
	fbNciAutomatic: 			FB_NciAutomatic;
	fbNciMdi: 					FB_NCI_MDI;
	F_TRIG1: 					F_TRIG;
	R_TRIG1: 					R_TRIG;
	nMode: 						WORD;
	fbSetOpModeSingleStep: 		FB_SetOpModeSingleStep;
	bSingleBlockAds: 			BOOL;
	fbConfirmMfunc: 			FB_ConfirmMfunc;
	nPrg: 						UINT;
	sTmpFile: 					STRING(255);
	sTmp: 						STRING;

	fbBlinker: 					FB_Blinker;
	fbWriteRParams: 			FB_WriteRParams;
	fbReadRParams:	 			FB_ReadRParams;	
	
	fbRTRIGReset:				R_TRIG;

END_VAR

(* ==========================================================*)
(*   FB: FB_NciChannel	                		             *)
(* ----------------------------------------------------------*)
(*   Desc: 													 *)
(*   Auth: MiB / TV                                          *)
(*   Date: 02.09.2005                                        *)
(*   Last: 02.04.2013                                        *)
(*   Rev.: 1.2                                               *)
(*	        1.1	20.07.2007 read and write of rParameters     *)
(* ==========================================================*)

IF bStateStop THEN
	bStateStart := FALSE;
END_IF

(* RESET *)
fbRTRIGReset(Clk := bStateReset);

IF fbRTRIGReset.Q THEN
	bStateStart := FALSE;
	bStateStop := FALSE;	
	ItpReset1.bExecute:= TRUE;	
END_IF



ItpReset1(sNciToPlc:= arrNCToPLC_NCIChannel_REF[nChan-1]);


(* M-Functions *)
PRG_GetFastMfunctions(nChan:= nChan );
fbConfirmMfunc(nChan:= nChan , bErr=> , nErrId=> );

(* Override *)
F_SetOverride(PLCFeedOverride, nChan, bFeedHold);

(* Skip Line *)
arrPLCToNC_NCIChannel_REF[nChan-1].SkipLine.0 := bPrgBlockIgnore;




(* OpModes *)
fbRTrigAuto( Clk := bModeAutomatic );
fbRTrigManual( Clk := bModeManual );
fbRTrigMDI( Clk := bModeMDI );
fbRTrigReference( Clk := bModeReference );




	(* ---------------------------------------------
	"NOT Ready"	// 0
	"Standby"	// 1 
	"Automatic"	// 2
	"MDI"			// 3
	"Manual"		// 4
	"Reference" // 5
	 ------------------------------------------------- *)

IF (fbRTrigAuto.Q) THEN
	bStateReset		:= TRUE;
	bModeReference := FALSE;
	bModeManual 	:= FALSE;
	bModeMDI 		:= FALSE;
 	bModeAutomatic  := TRUE;
	PLCNciChannelState.Mode[nChan] :=2;
END_IF

IF (fbRTrigMDI.Q) THEN
	bStateReset		:= TRUE;
	bModeReference := FALSE;
	bModeManual 	:= FALSE;
	bModeMDI 		:= TRUE;
  	bModeAutomatic := FALSE;
	PLCNciChannelState.Mode[nChan] :=3;
END_IF

IF (fbRTrigManual.Q) THEN
	bStateReset		:= TRUE;
	bModeReference := FALSE;
	bModeManual 	:= TRUE;
	bModeMDI 		:= FALSE;
 	bModeAutomatic := FALSE;
	PLCNciChannelState.Mode[nChan] :=4;
END_IF

IF (fbRTrigReference.Q) THEN
	bStateReset		:= TRUE;
	bModeReference := TRUE;
	bModeManual 	:= FALSE;
	bModeMDI 		:= FALSE;
 	bModeAutomatic := FALSE;
	PLCNciChannelState.Mode[nChan] :=5;
END_IF



(* SingleBlock *)
R_TRIG1(CLK:= bSingleBlock );
IF (R_TRIG1.Q) THEN
	bSingleBlockAds := TRUE;
	nMode := 16#01;				(* SingleStep Interpreter = 16#4000*)  (* Single Step NC Kern= 16#01 *)
END_IF

F_TRIG1(CLK:= bSingleBlock);
IF (F_TRIG1.Q) THEN
	bSingleBlockAds := TRUE;
	nMode := 16#0;
END_IF

IF bSingleBlockAds THEN
	fbSetOpModeSingleStep(
		nChan:= nChan,
		bExec:= bSingleBlockAds,
		nMode := nMode,
		bErr=> ,
		bBusy=> ,
		nErrId=> );
	IF NOT fbSetOpModeSingleStep.bBusy THEN
		bSingleBlockAds := FALSE;
		fbSetOpModeSingleStep(bExec := FALSE);
	END_IF
END_IF

IF bModeAutomatic THEN
	fbNciAutomatic(
		nChan:= nChan,
		bStateStop:= bStateStop,
		bStateStart:= bStateStart,
		sProgramName:= sProgramName);
END_IF

IF bModeMDI THEN
	nPrg := 10001 - nChan;               (* generate programm number for tmp MDI program; 9999.NC = channel1, 9998.NC = channel2, etc *)
	sTmpFile := 'C:\TwinCAT\CNC\';
	sTmpFile := CONCAT(sTmpFile, UINT_TO_STRING(nPrg));
	sTmpFile := CONCAT(sTmpFile,'.nc');

	fbNciMdi(
		bExec := NOT bStateReset,
		nChan:= nChan,
		sMDIString:= sMDIString ,
		sTmpFileName := sTmpFile,
		bStateStop:= bStateStop,
		bStateStart:= bStateStart);
END_IF


(* R-Parameter *)

(* example: read and write RParamter every second

	the paramters that are written to the NCI are defined in global Variables/Global_Nci/nRParamWrite[......
	the paramters that are read from the NCI are defined in global Variables/Global_Nci/nRParamRead[......

*)
fbBlinker(Taktzeit:= t#1s);

fbWriteRParams(
	bExec:= fbBlinker.Ausgang,
	nChan:= nChan);

fbReadRParams(
	bExec:= fbBlinker.Ausgang,
	nChan:= nChan);


IF (arrNCToPLC_NCIChannel_REF[nChan-1].ItpState =  NCI_INTERPRETER_IDLE OR arrNCToPLC_NCIChannel_REF[nChan-1].ItpState =  NCI_INTERPRETER_READY ) THEN
	ItpReset1.bExecute:= FALSE;	
	bStateReset := FALSE;
END_IF

//Add PiotrB
bStateError := arrNCToPLC_NCIChannel_REF[nChan-1].ErrorCode <> 0;

END_FUNCTION_BLOCK

// ---- POUs/Programy/Hbot/NCI/3_OPMODES/FB_NCIAutomatic.TcPOU
FUNCTION_BLOCK FB_NCIAutomatic
VAR_INPUT
	nChan: 						UINT;
	sProgramName: 				STRING(1024);
END_VAR
VAR_OUTPUT
END_VAR
VAR
	fbLoadStart: 				FB_LoadStart;
	ItpStartStop1: 				ItpStartStop;
	nItpState: 					UDINT;

	bCommandSingleStep: 		BOOL := FALSE;
	nItpMode: 					UDINT;
	bCommandLoadStart: 			BOOL := FALSE;
	bCommandEStop: 				BOOL := FALSE;
	bCommandEStopStepOn: 		BOOL := FALSE;
	fbEStop: 					FB_EStop;
	fbStepOnAfterEStop: 		FB_StepOnAfterEStop;
	sTmp: 						STRING;
END_VAR

VAR_IN_OUT
	bStateStart: 				BOOL;
	bStateStop: 				BOOL;
END_VAR

(* ==========================================================*)
(*   FB: FB_NciAutomatic		                             *)
(* ----------------------------------------------------------*)
(*   Desc:  										         *)
(*   Auth: MiB / TV                                          *)
(*   Date: 02.09.2005                                        *)
(*   Last: 02.04.2013                                        *)
(*   Rev.: 1.1                                               *)
(* ==========================================================*)

(* START, STOP, load program *)
nItpState	:=	arrNCToPLC_NCIChannel_REF[nChan-1].ItpState;
nItpMode 	:= arrNCToPLC_NCIChannel_REF[nChan-1].ItpMode;

IF (bStateStop) THEN				(* if STOP -> do not start anything *)
  bStateStart := FALSE;
END_IF

IF (nItpState = NCI_INTERPRETER_RUNNING AND nItpMode = 1 AND bStateStart) THEN
		bCommandSingleStep := TRUE;
END_IF

IF ( (nItpState = NCI_INTERPRETER_IDLE OR nItpState = NCI_INTERPRETER_READY) AND bStateStart) THEN
	bCommandLoadStart := TRUE;
END_IF

IF bStateStop THEN
	bCommandEStop := TRUE;
END_IF

IF bStateStart THEN
	bCommandEStopStepOn := TRUE;
END_IF

(* EStop programm *)
IF bCommandEStop THEN
	fbEStop(
		bExec:= TRUE,
		nChan:= nChan);
	IF NOT fbEStop.bBusy THEN
		fbEStop(bExec := FALSE);
		bCommandEStop := FALSE;
	END_IF
END_IF

(* Step on after EStop *)
IF bCommandEStopStepOn THEN
	fbStepOnAfterEStop(
		bExec:= TRUE,
		nChan:= nChan);
	IF NOT fbStepOnAfterEStop.bBusy THEN
		fbStepOnAfterEStop(bExec := FALSE);
		bCommandEStopStepOn := FALSE;
	END_IF
END_IF

(* load program and start it *)
IF bCommandLoadStart THEN
	fbLoadStart(
	bExec:= TRUE,
	sPrg:= sProgramName,
	nChan:= nChan,
	nErrId=> ,
	bBusy=> ,
	bErr=> );
	IF (NOT fbLoadStart.bBusy) THEN
		bCommandLoadStart := FALSE;
		fbLoadStart(bExec := FALSE);
	END_IF
END_IF


(* start single step *)
IF bCommandSingleStep THEN
	ItpStartStop1(
	bStart:= TRUE,
	bStop:= bStateStop,
	nChnId:= nChan,
	tTimeOut:= t#250ms,
	bBusy=> ,
	bErr=> ,
	nErrId=> );
	IF (NOT ItpStartStop1.bBusy) THEN
		ItpStartStop1(bStart:= FALSE, bStop := FALSE);
		bStateStop := FALSE;
		bCommandSingleStep := FALSE;
	END_IF
END_IF

bStateStart := FALSE;
bStateStop := FALSE;

END_FUNCTION_BLOCK

// ---- POUs/Programy/Hbot/NCI/1_CTRL/FB_LoadStart.TcPOU
FUNCTION_BLOCK FB_LoadStart
VAR_INPUT
	bExec: 			BOOL;
	sPrg: 			STRING(1024);
	nChan: 			UINT;
END_VAR
VAR_OUTPUT
	nErrId: 		UDINT;
	bBusy: 			BOOL;
	bErr:			BOOL;
END_VAR
VAR
	nState: 		UINT := 16#0;
	ItpLoadProg1: 	ItpLoadProgEx;
	ItpStartStop1:  ItpStartStopEx;
	nItpState: 		UDINT;
	fbRTrig: 		R_TRIG;
END_VAR

(* ==========================================================*)
(*     FB: FB_LoadStart			                             *)
(* ----------------------------------------------------------*)
(*   Desc: Load programm in NCI and after success start it	 *)
(*   Auth: MiB / TV                                          *)
(*   Date: 02.09.2005                                        *)
(*   Last: 02.04.2013                                        *)
(*   Rev.: 1.1                                               *)
(* ==========================================================*)



fbRTrig(Clk := bExec);

CASE nState OF
16#0:	(* init *)
		IF fbRTrig.Q THEN
			nItpState	:=	ItpGetStateInterpreter( arrNCToPLC_NCIChannel_REF[nChan-1] );
			IF nItpState = NCI_INTERPRETER_IDLE OR nItpState = NCI_INTERPRETER_READY THEN
				bBusy	:= TRUE;
				bErr	:= FALSE;
				nErrId	:= 0;
				nState := 16#10;
			ELSE
				nState := 16#30;   (* do nothing *)
			END_IF
		END_IF

16#10: (* load program *)

		ItpLoadProg1.bExecute:= TRUE;						
		ItpLoadProg1.sPrg:= sPrg;
		ItpLoadProg1.nLength:= LEN(sPrg);
		ItpLoadProg1.tTimeOut:= t#20s;
		nState	:= 16#15;		
16#15:
		IF (NOT ItpLoadProg1.bBusy) THEN
			ItpLoadProg1.bExecute := FALSE;
			IF NOT ItpLoadProg1.bErr THEN
				nState	:= 16#20;
			ELSE
				(* an error occured *)
				bErr		:= TRUE;
				nErrId	:= ItpLoadProg1.nErrId;
				nState	:= 16#999;
			END_IF
		END_IF

16#20: (* start program *)

		ItpStartStop1.bStart := TRUE;
		ItpStartStop1.bStop := FALSE;				
		ItpStartStop1.tTimeOut:= T#250MS;		
		nState := 16#25; 	
16#25:

		IF (NOT ItpStartStop1.bBusy) THEN
			ItpStartStop1.bStart:=FALSE;
			IF NOT ItpStartStop1.bErr THEN
				nState := 16#30; (* end *)
			ELSE
			(* an error occured *)
				bErr		:= TRUE;
				nErrId	:= ItpStartStop1.nErrId;
				nState	:= 16#999;
			END_IF
		END_IF

16#30:

		bBusy := FALSE;
		bErr	:= FALSE;
		nErrId	:= 0;
		nState := 0;


16#999:	(* Error *)
		bBusy := FALSE;
		nState := 0;

END_CASE

ItpStartStop1( sNciToPlc := arrNCToPLC_NCIChannel_REF[nChan-1]);	
ItpLoadProg1( sNciToPlc := arrNCToPLC_NCIChannel_REF[nChan-1]);

END_FUNCTION_BLOCK

// ---- POUs/Programy/Hbot/NCI/1_CTRL/FB_EStop.TcPOU
FUNCTION_BLOCK FB_EStop
VAR_INPUT
	bExec: 		BOOL;
	nChan: 		UINT;
END_VAR
VAR_OUTPUT
	bBusy: 		BOOL;
	nErrId: 		UDINT;
	bErr: 		BOOL;
END_VAR
VAR
	fbRTrig: 	R_TRIG;
	nState: 		UINT;
	fbADSREAD: 	ADSREAD;
	nGroup: 		UDINT;
	fbItpEStop: ItpEStopEx;
END_VAR

(* ==========================================================*)
(*     FB: FB_EStop					                         *)
(* ----------------------------------------------------------*)
(*   Desc:                                                   *)
(*   Auth: MiB  / TV                                         *)
(*   Date: 02.09.2005                                        *)
(*   Last: 02.04.2013                                        *)
(*   Rev.: 1.1                                               *)
(* ==========================================================*)


fbRTrig(Clk := bExec);

CASE nState OF


16#0: (* init *)
		IF fbRTrig.Q THEN
			bBusy	:= TRUE;
			bErr	:= FALSE;
			nErrId	:= 0;
			nState := 16#10;
		END_IF

16#10: (* Read Group ID *)
		fbADSREAD(
			NETID:= ,
			PORT:= 	501,  			(* NCI Channel *)
			IDXGRP:= 16#2000+nChan, (* Spezifikation für Kanal-Parameter *)
			IDXOFFS:=16#21 ,			(* 0x00000021  Read  every  UINT32  1   Gruppen-ID (nur eindeutig für 3D- und FIFO-Kanal   *)
			LEN:= SIZEOF(nGroup),
			DESTADDR:=ADR(nGroup) ,
			READ:= TRUE,
			TMOUT:= T#200ms,
			BUSY=> ,
			ERR=> ,
			ERRID=> );

		IF fbADSREAD.ERR THEN
			fbADSREAD(READ := FALSE);
			bErr := TRUE;
			nErrId := fbADSREAD.ERRID;
			nState := 16#999;
		END_IF

		IF (NOT fbADSREAD.ERR) AND (NOT fbADSREAD.BUSY) THEN
			fbADSREAD(READ := FALSE);
			nState := 16#20;
		END_IF;

16#20: (* initiate EStop in NCI *)
		fbItpEStop.bExecute := TRUE;
		fbItpEStop.tTimeOut:= T#250MS;
		nState := 16#25;		
16#25:			
		IF NOT fbItpEStop.bBusy THEN
			fbItpEStop.bExecute := FALSE;
			IF fbItpEStop.bErr THEN
				nErrId := fbItpEStop.nErrId;
				bErr := TRUE;
				nState := 16#999;
			ELSE
				nState := 16#0;
				bBusy := FALSE;
			END_IF
		END_IF

16#999:	(* Error *)
		bBusy := FALSE;
		nState := 0;
END_CASE

fbItpEStop( sNciToPlc := arrNCToPLC_NCIChannel_REF[nChan-1]);

END_FUNCTION_BLOCK

// ---- POUs/Programy/Hbot/NCI/1_CTRL/FB_StepOnAfterEStop.TcPOU
FUNCTION_BLOCK FB_StepOnAfterEStop
VAR_INPUT
	bExec: 						BOOL;
	nChan: 						UINT;
END_VAR
VAR_OUTPUT
	bBusy: 						BOOL;
	nErrId: 						UDINT;
	bErr: 						BOOL;
END_VAR
VAR
	fbRTrig: 					R_TRIG;
	nState: 						UINT;
	fbADSREAD: 					ADSREAD;
	nGroup: 						UDINT;
	fbItpStepOnAfterEStop: 	ItpStepOnAfterEStop;
END_VAR

(* ==========================================================*)
(*     FB: FB_StepOnAfterEStop	                             *)
(* ----------------------------------------------------------*)
(*   Desc:                                                   *)
(*   Auth: MiB / TV                                          *)
(*   Date: 02.09.2005                                        *)
(*   Last: 02.04.2013                                        *)
(*   Rev.: 1.1                                               *)
(* ==========================================================*)

fbRTrig(Clk := bExec);

CASE nState OF
16#0: (* init *)
		IF fbRTrig.Q THEN
			bBusy	:= TRUE;
			bErr	:= FALSE;
			nErrId	:= 0;
			nState := 16#10;
		END_IF

16#10: (* Read Group ID *)
		fbADSREAD(
			NETID:= ,
			PORT:= 	501,  			(* NCI Channel *)
			IDXGRP:= 16#2000+nChan, (* Spezifikation für Kanal-Parameter *)
			IDXOFFS:=16#21 ,			(* 0x00000021  Read  every  UINT32  1   Gruppen-ID (nur eindeutig für 3D- und FIFO-Kanal   *)
			LEN:= SIZEOF(nGroup),
			DESTADDR:=ADR(nGroup) ,
			READ:= TRUE,
			TMOUT:= T#200ms,
			BUSY=> ,
			ERR=> ,
			ERRID=> );
		IF NOT fbADSREAD.BUSY THEN
			fbADSREAD(READ := FALSE);
			IF fbADSREAD.ERR THEN
				fbADSREAD(READ := FALSE);
				bErr := TRUE;
				nErrId := fbADSREAD.ERRID;
				nState := 16#999;
			ELSE
				nState := 16#20;
			END_IF
		END_IF

16#20: (* initiate Step on after EStop in NCI *)
		fbItpStepOnAfterEStop(
			bExecute:= TRUE,
			nGrpId:= nGroup,
			tTimeOut:= t#250ms);
		IF NOT fbItpStepOnAfterEStop.bBusy THEN
			fbItpStepOnAfterEStop(bExecute := FALSE);
			IF fbItpStepOnAfterEStop.bErr THEN
				nErrId := fbItpStepOnAfterEStop.nErrId;
				bErr := TRUE;
				nState := 16#999;
			ELSE
				nState := 16#0;
				bBusy := FALSE;
			END_IF
		END_IF


16#999:	(* Error *)
		bBusy := FALSE;
		nState := 0;

END_CASE

END_FUNCTION_BLOCK

// ---- POUs/Programy/Hbot/NCI/3_OPMODES/FB_NCI_MDI.TcPOU
FUNCTION_BLOCK FB_NCI_MDI
VAR_INPUT
	sMDIString: 		STRING(1024);
	sTmpFileName:		STRING(255);
	nChan: 				UINT;
	bExec:				BOOL;
END_VAR
VAR_OUTPUT
	nErrId: 				UDINT;
	bErr:					BOOL;
END_VAR
VAR
	nState: 				UINT;
	hFile: 				UINT;
	fbFileOpen: 		FB_FileOpen;
	fbFilePuts: 		FB_FilePuts;
	fbFileClose: 		FB_FileClose;

	fbLoadStart: 		FB_LoadStart;
	fbItpStartStop: 	ItpStartStopEx;
	fbItpEStop:			FB_EStop;
	fbItpIsEStop:		ItpIsEStop;
	nGroup:				UDINT;
	fbADSREAD: 			ADSREAD;
	fbStepOnAfterEStop: FB_StepOnAfterEStop;

	fbRtrigInit: 		R_TRIG;
	nItpState: 			UDINT;
	bCommandStart: 	BOOL;
	bCommandStop: 		BOOL;
END_VAR

VAR_IN_OUT
	bStateStop: 		BOOL;
	bStateStart: 		BOOL;
END_VAR

(* ==========================================================*)
(*   FB: FB_NciMdi		              		                 *)
(* ----------------------------------------------------------*)
(*   Desc: create file from sMDIString and handle start/stop *)
(*   Auth: MiB / TV                                          *)
(*   Date: 02.09.2005                                        *)
(*   Last: 02.04.2013                                        *)
(*   Rev.: 1.2	                                             *)
(*			  20.12.2005 CL added continuing of MDI processafter*)
(*							 stop							 *)
(* ==========================================================*)


(* rising edge detection Init *)
fbRtrigInit(Clk := bExec);

IF bStateStart THEN
	bCommandStart := TRUE;
END_IF

IF bStateStop THEN
	bCommandStop := TRUE;
	bCommandStart := FALSE;
END_IF

bStateStart := FALSE;
bStateStop := FALSE;


CASE nState OF

16#0: (* init *)
	IF fbRtrigInit.Q THEN
		bErr := FALSE;
		nErrId := 0;
		nState := 16#5;
	END_IF

16#5: (* Read Group ID *)
		fbADSREAD(
			NETID:= ,
			PORT:= 	501,  			(* NCI Channel *)
			IDXGRP:= 16#2000+nChan, (* Spezifikation für Kanal-Parameter *)
			IDXOFFS:=16#21 ,			(* 0x00000021  Read  every  UINT32  1   Gruppen-ID (nur eindeutig für 3D- und FIFO-Kanal   *)
			LEN:= SIZEOF(nGroup),
			DESTADDR:=ADR(nGroup) ,
			READ:= TRUE,
			TMOUT:= T#200ms,
			BUSY=> ,
			ERR=> ,
			ERRID=> );

		IF fbADSREAD.ERR THEN
			fbADSREAD(READ := FALSE);
			bErr := TRUE;
			nErrId := fbADSREAD.ERRID;
			nState := 16#999;
		END_IF

		IF (NOT fbADSREAD.ERR) AND (NOT fbADSREAD.BUSY) THEN
			fbADSREAD(READ := FALSE);
			nState := 16#10;
		END_IF;

16#10: (* wait for start *)
	IF bCommandStart THEN
		nState := 16#20;
		bCommandStart := FALSE;
		IF  sTmpFileName='' THEN
			sTmpFileName := 'C:\TwinCAT\CNC\9999.nc'; (* standard filename for MDI *)
		END_IF
	END_IF;


16#20:	(* create file *)
   fbFileOpen(
		sNetId:= '',
		sPathName:= sTmpFileName,
		nMode:= FOPEN_MODEWRITE OR FOPEN_MODETEXT,
		ePath:= PATH_GENERIC,
		bExecute:= TRUE,
		tTimeout:= T#1s,
		hFile=> hFile);
	IF NOT fbFileOpen.bBusy THEN
		fbFileOpen(bExecute := FALSE);
		IF fbFileOpen.bError THEN
			nErrId := fbFileOpen.nErrId;
			nState := 16#999;
		ELSE
			nState := 16#30;
		END_IF
	END_IF

16#30: (* put MDI String into file *)
	fbFilePuts(
		sNetId:= '',
		hFile:= hFile,
		sLine:= sMDIString,
		bExecute:= TRUE,
		tTimeout:= t#1s);
	IF NOT fbFilePuts.bBusy THEN
		fbFilePuts(bExecute := FALSE);
		IF fbFilePuts.bError THEN
			nErrId := fbFilePuts.nErrId;
			nState := 16#999;
		ELSE
			nState := 16#40;
		END_IF
	END_IF

16#40:  (* append @714 (= Dekodierstop) *)
	fbFilePuts(
		sNetId:= '',
		hFile:= hFile,
		sLine:= '$0A@714$0A',
		bExecute:= TRUE,
		tTimeout:= t#1s);
	IF NOT fbFilePuts.bBusy THEN
		fbFilePuts(bExecute := FALSE);
		IF fbFilePuts.bError THEN
			nErrId := fbFilePuts.nErrId;
			nState := 16#999;
		ELSE
			nState := 16#50;
		END_IF
	END_IF

16#50:	(* close file *)
	fbFileClose(
		sNetId:= '',
		hFile:= hFile,
		bExecute:= TRUE,
		tTimeout:= t#1s);
	IF NOT fbFileClose.bBusy THEN
		fbFileClose(bExecute := FALSE);
		IF fbFileClose.bError THEN
			nErrId := fbFileClose.nErrId;
			nState := 16#999;
		ELSE
			nState := 16#60;
		END_IF
	END_IF

16#60: (* load and start program *)
	fbLoadStart(
		bExec:= TRUE,
		sPrg:= sTmpFileName,
		nChan:= nChan);
	IF NOT fbLoadStart.bBusy THEN
		fbLoadStart(bExec := FALSE);
		IF fbLoadStart.bErr THEN
			nErrId := fbLoadStart.nErrId;
			nState := 16#999;
		ELSE
			nState := 16#70;
		END_IF
	END_IF

16#70: (* wait for end of program and handle stop *)
		IF (bCommandStop) THEN
			(*fbItpStartStop(
				bStart:= FALSE,
				bStop:= TRUE,
				nChnId:= nChan,
				tTimeOut:= T#250ms);
			IF NOT fbItpStartStop.bBusy THEN
				fbItpStartStop(bStop := FALSE, bStart := FALSE);
				bCommandStop := FALSE;
			END_IF*)
			fbItpEStop(
				bExec:= TRUE,
				nChan:= nChan);
			IF NOT fbItpEStop.bBusy THEN
				fbItpEStop(bExec := FALSE);
				bCommandStop := FALSE;
			END_IF
		END_IF

		fbItpIsEStop(
   		bExecute:=   TRUE,
   		nGrpId:=     nGroup,
   		tTimeOut:=   t#250ms);
		IF NOT fbItpIsEStop.bBusy THEN
			IF fbItpIsEStop.bEStop THEN
				nState := 16#80;
			END_IF
			fbItpIsEStop(bExecute:= FALSE);
		END_IF

		nItpState := ItpGetStateInterpreter( arrNCToPLC_NCIChannel_REF[nChan-1] );
		IF nItpState = NCI_INTERPRETER_IDLE OR nItpState = NCI_INTERPRETER_READY OR nItpState = NCI_INTERPRETER_ABORTED THEN
			nState := 16#10;
		END_IF

16#80: (* waiting for continue *)
		IF bCommandStart THEN
			fbStepOnAfterEStop(
				bExec:= TRUE,
				nChan:= nChan);
			IF NOT fbStepOnAfterEStop.bBusy THEN
				fbStepOnAfterEStop(bExec := FALSE);
				bCommandStart := FALSE;
				nState:= 16#70;
			END_IF
		END_IF

		bCommandStop := FALSE; (* we are in stop already *)
		nItpState := ItpGetStateInterpreter( arrNCToPLC_NCIChannel_REF[nChan-1] );
		IF nItpState = NCI_INTERPRETER_IDLE OR nItpState = NCI_INTERPRETER_READY OR nItpState = NCI_INTERPRETER_ABORTED THEN
			nState := 16#10;
		END_IF

16#999:   (* error *)
		bErr := TRUE;
	   nState := 16#0;   (* init *)

END_CASE

END_FUNCTION_BLOCK

// ---- POUs/Programy/Hbot/NCI/1_CTRL/FB_SetOpModeSingleStep.TcPOU
FUNCTION_BLOCK FB_SetOpModeSingleStep
VAR_INPUT
	nChan: 		UINT;
	bExec: 		BOOL;
	nMode: 		WORD;
END_VAR
VAR_OUTPUT
	bErr:		BOOL;
	bBusy: 		BOOL;
	nErrId: 	UDINT;
END_VAR
VAR
	nState: 		UINT;
	fbRtrig: 	R_TRIG;
	fbAdsWrite: ADSWRITE;
END_VAR

(* ==========================================================*)
(*     FB: FB_SetOpMode 			                         *)
(* ----------------------------------------------------------*)
(*   Desc:                                                   *)
(*   Auth: MiB / TV                                          *)
(*   Date: 02.09.2005                                        *)
(*   Last: 02.04.2013                                        *)
(*   Rev.: 1.1                                               *)
(* ==========================================================*)


fbRtrig(Clk := bExec);


CASE nState OF
16#0: (* init *)
		IF fbRtrig.Q THEN
			bBusy	:= TRUE;
			bErr	:= FALSE;
			nErrId	:= 0;
			nState := 16#10;
		END_IF

16#10: (* single block *)
		fbAdsWrite(
			NETID:= ,
			PORT:= 501,						(* NCI *)
			IDXGRP:= 16#2200 + nChan,  (* Spezifikation für Kanal-Funktionen  *)
			IDXOFFS:= 16#5 ,				(* Setze Interpreter Betriebsart			*)
			LEN:= SIZEOF(nMode),
			SRCADDR:= ADR(nMode),
			WRITE:= TRUE,
			TMOUT:= T#200ms,
			BUSY=> ,
			ERR=> ,
			ERRID=> );
		IF NOT fbAdsWrite.BUSY THEN
			fbAdsWrite(WRITE := FALSE);
			IF fbAdsWrite.ERR THEN
				bErr := TRUE;
				nErrId := fbAdsWrite.ERRID;
				nState := 16#999;
			ELSE
				nState := 16#20;
			END_IF
		END_IF

16#20: (* ready *)
		bBusy := FALSE;
		bErr	:= FALSE;
		nErrId	:= 0;
		nState := 0;

16#999:	(* Error *)
		bBusy := FALSE;
		nState := 0;


END_CASE

END_FUNCTION_BLOCK

// ---- POUs/Programy/Hbot/NCI/1_CTRL/FB_ConfirmMFunc.TcPOU
FUNCTION_BLOCK FB_ConfirmMFunc
VAR_INPUT
	nChan: 		UINT;
END_VAR
VAR_OUTPUT
	bErr: 		BOOL;
	nErrId: 	UDINT;
END_VAR
VAR
	fbConfirm: 	ItpConfirmHsk;
	bConfirm:	BOOL := FALSE;
	nAktMfunc:	INT :=  -1;
	TON1: 		TON;
	i: UINT;
END_VAR

(* ==========================================================*)
(*     FB: FB_ConfirmMfunc			                         *)
(* ----------------------------------------------------------*)
(*   Desc:                                                   *)
(*   Auth: MiB / TV                                          *)
(*   Date: 25.04.2006                                        *)
(*   Last: 02.04.2013                                        *)
(*   Rev.: 2.1                                              *)
(* ==========================================================*)



(* check for m function and store information in bMFunc Array *)

	IF ItpIsHskMFunc(arrNCToPLC_NCIChannel_REF[nChan-1] ) THEN
		nAktMfunc := ItpGetHskMFunc(arrNCToPLC_NCIChannel_REF[nChan-1]);
		bMFunc[nChan-1, nAktMfunc] := TRUE;
	ELSE
		nAktMfunc := -1;
		bConfirm := FALSE;
		FOR i := 0 TO 159 DO
			bMFunc[nChan-1, i] := FALSE;
			bQuitMFunc[nChan-1, i] := FALSE;
		END_FOR
	END_IF


(* confirm m function, if bit in array bQuitMFunc is set *)
	IF (nAktMfunc <> -1) THEN
		IF bQuitMFunc[nChan-1, nAktMfunc] THEN
			bConfirm := TRUE;
		END_IF
		bQuitMFunc[nChan-1,nAktMfunc] := FALSE;
	END_IF


fbConfirm(
		bExecute := bConfirm,
		sNciToPlc:= arrNCToPLC_NCIChannel_REF[nChan-1],
		sPlcToNci:= arrPLCToNC_NCIChannel_REF[nChan-1]
			);

END_FUNCTION_BLOCK

// ---- POUs/Programy/Hbot/NCI/Util/FB_Blinker.TcPOU
FUNCTION_BLOCK FB_Blinker
VAR_INPUT
	Taktzeit: TIME;
END_VAR
VAR_OUTPUT
	Ausgang: BOOL;
END_VAR
VAR
	Timer1: TON;
END_VAR

Timer1(In := NOT Timer1.Q, PT := Taktzeit);
Ausgang := Taktzeit/2 > Timer1.ET;

END_FUNCTION_BLOCK

// ---- POUs/Programy/Hbot/NCI/9_MISC/FB_WriteRParams.TcPOU
FUNCTION_BLOCK FB_WriteRParams
VAR_INPUT
	bExec: 						BOOL;
	bBusy: 						BOOL;
	nChan: 						UINT;
END_VAR
VAR_OUTPUT
	nErrId: 					UDINT;
	bErr: 						BOOL;
END_VAR
VAR
	fbWriteRParams: 			ItpWriteRParams;
	nIndex: 					DINT;
	nCount: 					DINT;
END_VAR

(* ==========================================================*)
(*   PRG: FB_WriteRParams			        		            	 *)
(* ----------------------------------------------------------*)
(*   Desc:  writes the R-Parameter from global					 *)
(*				array nRParamWrite to the NCI 					    *)
(*   Auth: MiB                                               *)
(*   Date: 20.07.2007                               	       *)
(*   Rev.: 1.0                                               *)
(* ==========================================================*)


nIndex := nStartIndexWriteRParam;
nCount := (nEndIndexWriteRParm - nStartIndexWriteRParam) + 1;


fbWriteRParams(
	bExecute:= bExec,
	nChnId:= nChan ,
	pAddr:= ADR(nRParamWrite[nChan - 1, nStartIndexWriteRParam]),
	nIndex:= nIndex,
	nCount:= nCount,
	tTimeOut:= t#2s,
	bBusy=> bBusy,
	bErr=> bErr,
	nErrId=>nErrId );

END_FUNCTION_BLOCK

// ---- POUs/Programy/Hbot/NCI/9_MISC/FB_ReadRParams.TcPOU
FUNCTION_BLOCK FB_ReadRParams
VAR_INPUT
	bExec: 						BOOL;
	bBusy: 						BOOL;
	nChan: 						UINT;
END_VAR
VAR_OUTPUT
	nErrId: 					UDINT;
	bErr: 						BOOL;
END_VAR
VAR
	fbReadRParams: 				ItpReadRParams;
END_VAR

(* ==========================================================*)
(*   PRG: FB_ReadRParams			        		            	 *)
(* ----------------------------------------------------------*)
(*   Desc:  reads the R-Parameter from the NCI and 			 *)
(*				store ist in global array nRParamRead 			    *)
(*   Auth: MiB                                               *)
(*   Date: 20.07.2007                               	       *)
(*   Rev.: 1.0                                               *)
(* ==========================================================*)


fbReadRParams(
	bExecute:= bExec,
	nChnId:= nChan,
	pAddr:= ADR(nRParamRead[nChan - 1, nStartIndexReadRParam]),
	nIndex:= nStartIndexReadRParam,
	nCount:= (nEndIndexReadRParam - nStartIndexReadRParam) + 1,
	tTimeOut:= t#2s,
	bBusy=> bBusy,
	bErr=> bErr,
	nErrId=>nErrId );

END_FUNCTION_BLOCK

// ---- POUs/Programy/Hbot/NCI/9_MISC/PRG_GetFastMFunctions.TcPOU
PROGRAM PRG_GetFastMFunctions
VAR_INPUT
	nChan: 	UINT;
END_VAR
VAR
	i: 		UINT;
	l: 		SINT;
	bBit: 	BOOL;
	index: 	UINT;
END_VAR

(* ==========================================================*)
(*   PRG: P_GetFastMfunctions		        		            	 *)
(* ----------------------------------------------------------*)
(*   Desc: fill the global defined M-functions Array with    *)
(*			  fast M-Functions from NCI Channel                 *)
(*   Auth: MiB                                               *)
(*   Date: 02.09.2005                                        *)
(*   Rev.: 1.0                                               *)
(* ==========================================================*)



IF (nChan<2) THEN   (* NCI channel starts at 2 *)
	RETURN;
END_IF;

FOR i:=0 TO 4 DO  (* check all 5 dwords *)
	FOR l := 0 TO 31 DO
		bBit := GETBIT32(arrNCToPLC_NCIChannel_REF[nChan-1].FastMFuncMask[i+1], l);
      index := (i*32) + l;
		IF ( bBit ) THEN
			bfastMFunc[nChan-1,index] := TRUE;
		ELSE
			bfastMFunc[nChan-1,index] := FALSE;
		END_IF
	END_FOR
END_FOR

END_PROGRAM

// ---- POUs/Programy/Hbot/NCI/1_CTRL/F_SetOverride.TcPOU
FUNCTION F_SetOverride : BOOL
VAR_INPUT
	nOverride: 	UDINT;
	nChannel: 	UINT;
	bFeedHold: 	BOOL;
END_VAR

(* ==========================================================*)
(*   FUN: F_SetOverride			                           	 *)
(* ----------------------------------------------------------*)
(*   Desc:                                                   *)
(*   Auth: MiB / TV                                          *)
(*   Date: 02.09.2005                                        *)
(*   Last: 02.04.2013                                        *)
(*   Rev.: 1.1                                               *)
(*    1.1 25.4.2006: bFeedHold rausgenommen	(MiB)		 *)
(* 1.2 12.8.2008: FeedHold aus PLCMachineMode reingenommen *)
(* ==========================================================*)


(* channl 1 = PTP channel *)

(* NCI channels *)
IF (nChannel > 1) THEN
		IF (NOT PLCMachineMode[nChannel].FeedHold) THEN
			ItpSetOverridePercent(nOverride, arrPLCToNC_NCIChannel_REF[nChannel-1]);
		ELSE
			ItpSetOverridePercent(0, arrPLCToNC_NCIChannel_REF[nChannel-1]);
		END_IF
END_IF

F_SetOverride := TRUE;

END_FUNCTION

// ---- POUs/Programy/Hbot/NCI/2_GROUPS/PRG_GroupAxesToNCI.TcPOU
PROGRAM PRG_GroupAxesToNCI
VAR_INPUT
	stMachineMode 	: ST_MachineMode;
	nChan : UINT;
END_VAR
VAR
	fbTrigBuildGroup	: 	R_TRIG;
	fbTrigReleaseGroup	: 	R_TRIG;
	fbBuildGroup1		: 	FB_BuildGroup;
	fbReleaseGroup1		: 	FB_ReleaseGroup;
	bGroup1Release		: 	BOOL := FALSE;
	nState 				:	UINT;
	bBuildGroup			: 	BOOL;
	bClearGroup			: 	BOOL;
END_VAR

VAR_IN_OUT
	stAxisRef_X			: Axis_REF;
	stAxisRef_Y			: Axis_REF;
END_VAR

(* ==========================================================*)
(*   PRG: GroupAxisToNci			        		         *)
(* ----------------------------------------------------------*)
(*   Desc: 													 *)
(*   Auth: MiB / TV                                          *)
(*   Date: 02.09.2005                                        *)
(*   Last: 02.04.2013                                        *)
(*   Rev.: 1.1                                               *)
(* ==========================================================*)


(* build axis3d groups *)

(* homing status of 1st group *)
nChan := GVL_NCI.nChan;
bBuildGroup := stMachineMode.Automatic OR stMachineMode.MDI;			(* this is an example condition for building a group *)
bClearGroup := stMachineMode.Homing OR stMachineMode.Manual;		(* this is an exmaple condition for releasing a group *)

IF (nState = 0) THEN
	fbTrigBuildGroup( clk := bBuildGroup );
	IF fbTrigBuildGroup.Q THEN
		bGroup1 := TRUE;
		bGroup1Release := FALSE;
		nState := 0;
	
	END_IF
	
	fbTrigReleaseGroup( clk := (bClearGroup) );
	IF fbTrigReleaseGroup.Q THEN
		bGroup1 := FALSE;
		bGroup1Release := TRUE;
		nState := 0;
	END_IF
END_IF

CASE nState OF

0: (* Wait for action *)
	IF bGroup1 OR bGroup1Release THEN
		nState := nState + 1;
	END_IF

1: (* Reset axis *)
	(*PRG_ResetAllAxesWithError(execute := TRUE);
	IF PRG_ResetAllAxesWithError.Done THEN*)
		IF bGroup1 THEN   (* buid group *)
			nState := 10;
		END_IF;
		IF bGroup1Release THEN
			nState := 20;	(* release group *)
		END_IF

	(*END_IF*)


10:(* build 1st group in channel2 *)
	fbBuildGroup1(
		bExec:= bGroup1 ,
		nChan:= nChan,
		nXAxisId:= stAxisRef_X.NcToPlc.AxisId,
		nYAxisId:= stAxisRef_Y.NcToPlc.AxisId,
		nZAxisId:= ,
		nQ1AxisId:= ,
		nQ2AxisId:= ,
		nQ3AxisId:= ,
		nQ4AxisId:= ,
		nQ5AxisId:= ,
		nGroup => nGroup[nChan-1],
		bBusy=> ,
		bErr=> ,
		nErrId=> );



	IF (NOT fbBuildGroup1.bBusy) AND NOT fbBuildGroup1.bErr AND bGroup1 (*AND (NOT fbBuildGroup2.bBusy) AND NOT fbBuildGroup2.bErr AND bGroup2 *) THEN
		fbBuildGroup1( bExec := FALSE );
		bGroup1 := FALSE;
		nState := 0;
	END_IF

	IF ((NOT fbBuildGroup1.bBusy) AND fbBuildGroup1.bErr)  THEN
		fbBuildGroup1( bExec := FALSE );
		bGroup1 := TRUE;   (*bei Fehler nochmal versuchen *)
		nState := 0;
	END_IF


20: (* release Group *)
			fbReleaseGroup1(
			bExec:= bGroup1Release,
			nChan:= nChan);
		IF (NOT fbReleaseGroup1.bBusy) AND NOT fbReleaseGroup1.bErr  AND bGroup1Release THEN
			fbReleaseGroup1( bExec := FALSE );
			bGroup1Release := FALSE;
			nState := 0;
		END_IF

		IF (NOT fbReleaseGroup1.bBusy) AND fbReleaseGroup1.bErr THEN
			fbReleaseGroup1( bExec := FALSE );
			bGroup1Release := TRUE; (* bei Fehler weiter versuchen, Gruppe aufzulösen *)
			nState := 0;
		END_IF
END_CASE

END_PROGRAM

// ---- POUs/Programy/Hbot/NCI/2_GROUPS/FB_BuildGroup.TcPOU
FUNCTION_BLOCK FB_BuildGroup
VAR_INPUT
	bExec: 			BOOL;
	nChan:			UINT;
	nXAxisId:		DWORD;
	nYAxisId:		DWORD;
	nZAxisId:		DWORD;
	nQ1AxisId:		DWORD;
	nQ2AxisId:		DWORD;
	nQ3AxisId:		DWORD;
	nQ4AxisId:		DWORD;
	nQ5AxisId:		DWORD;
END_VAR

VAR_OUTPUT
	nGroup:			UDINT;
	bBusy: 			BOOL;
	bErr: 			BOOL;
	nErrId:			UDINT:=0;
END_VAR
VAR
	nState: 			UINT:=0;
	ADSREAD1: 		ADSREAD;
	fbClearGrp: 	CfgReconfigGroup;
	fbBuildGrp: 	CfgBuildExt3DGroup;
	fbRtrig: 		R_TRIG;
END_VAR

(* ==========================================================*)
(*   FB: FB_BuildGroup			                             *)
(* ----------------------------------------------------------*)
(*   Desc: Build 3-d Group                                   *)
(*   Auth: MiB                                               *)
(*   Date: 02.09.2005                                        *)
(*   Last: 02.04.2013                                        *)
(*   Rev.: 1.1                                               *)
(* ==========================================================*)


fbRtrig(Clk := bExec);

CASE nState OF
16#0: (* init *)
		IF fbRtrig.Q THEN
			bBusy	:= TRUE;
			bErr	:= FALSE;
			nErrId	:= 0;
			nState := 16#10;
		END_IF


16#10: (* Read Group ID *)
		ADSREAD1(
			NETID:= ,
			PORT:= 	501,  			(* NCI Channel *)
			IDXGRP:= 16#2000+nChan, (* Spezifikation für Kanal-Parameter *)
			IDXOFFS:=16#21 ,			(* 0x00000021  Read  every  UINT32  1   Gruppen-ID (nur eindeutig für 3D- und FIFO-Kanal   *)
			LEN:= SIZEOF(nGroup),
			DESTADDR:=ADR(nGroup) ,
			READ:= TRUE,
			TMOUT:= T#200ms,
			BUSY=> ,
			ERR=> ,
			ERRID=> );

		IF ADSREAD1.ERR THEN
			bErr := TRUE;
			nErrId := ADSREAD1.ERRID;
			nState := 16#999;
		END_IF

		IF (NOT ADSREAD1.ERR) AND (NOT ADSREAD1.BUSY) THEN
			ADSREAD1(READ := FALSE);
			nState := 16#20;
		END_IF;

16#20: (* clear old interpolation Group *)

	fbClearGrp(
		bExecute:= TRUE,
		nGroupId:= nGroup,
		tTimeOut:= T#200ms);

	IF NOT fbClearGrp.bBusy THEN
		fbClearGrp(bExecute:= FALSE);
		IF NOT fbClearGrp.bErr THEN
			nState	:= 16#30;
		ELSE
			(* an error occured *)
			bErr		:= TRUE;
			nErrId	:= fbClearGrp.nErrId;
			nState	:= 16#999;
		END_IF
	END_IF

16#30: (* build new interploation group *)
	fbBuildGrp(
		bExecute	:= TRUE ,
		nGroupId	:= nGroup,
		nXAxisId	:= nXAxisId,
		nYAxisId	:= nYAxisId,
		nZAxisId :=	nZAxisId,
		nQ1AxisId:= nQ1AxisId,
		nQ2AxisId:= nQ2AxisId,
		nQ3AxisId:= nQ3AxisId,
		nQ4AxisId:= nQ4AxisId,
		nQ5AxisId:= nQ5AxisId,
		tTimeOut:= T#200ms);


	IF NOT fbBuildGrp.bBusy THEN
		fbBuildGrp( bExecute := FALSE );
		IF NOT fbBuildGrp.bErr THEN
			nState	:= 16#40;
		ELSE
			(* an error occured *)
			bErr		:= TRUE;
			nErrId	:= fbBuildGrp.nErrId;
			nState	:= 16#999;
		END_IF
	END_IF

16#40: (* end *)
	bBusy := FALSE;
	nState := 0;


16#999:	(* Error *)
		bBusy := FALSE;
		nState := 0;

END_CASE

END_FUNCTION_BLOCK

// ---- POUs/Programy/Hbot/NCI/2_GROUPS/FB_ReleaseGroup.TcPOU
FUNCTION_BLOCK FB_ReleaseGroup
VAR_INPUT
	bExec: 			BOOL;
	nChan:			UINT;
END_VAR

VAR_OUTPUT
	bBusy: 			BOOL;
	bErr: 			BOOL;
	nErrId:			UDINT:=0;
END_VAR
VAR
	nState: 			UINT:=0;
	fbAdsRead: 		ADSREAD;
	nGroup:			UDINT;
	fbClearGrp: 	CfgReconfigGroup;
	fbRtrig: 		R_TRIG;
END_VAR

(* ==========================================================*)
(*   FB: FB_ReleaseGroup		                             *)
(* ----------------------------------------------------------*)
(*   Desc: Release all axis from group		                 *)
(*   Auth: MiB / TV                                          *)
(*   Date: 02.09.2005                                        *)
(*   Last: 02.04.2013                                        *)
(*   Rev.: 1.2                                               *)
(* ==========================================================*)

fbRtrig(Clk := bExec);


CASE nState OF
16#0: (* init *)
		IF fbRtrig.Q THEN
			bBusy	:= TRUE;
			bErr	:= FALSE;
			nErrId	:= 0;
			nState := 16#10;
		END_IF


16#10: (* Read Group ID *)
		fbAdsRead(
			NETID:= ,
			PORT:= 	501,  			(* NCI Channel *)
			IDXGRP:= 16#2000+nChan, (* Spezifikation für Kanal-Parameter *)
			IDXOFFS:=16#21 ,			(* 0x00000021  Read  every  UINT32  1   Gruppen-ID (nur eindeutig für 3D- und FIFO-Kanal   *)
			LEN:= SIZEOF(nGroup),
			DESTADDR:=ADR(nGroup) ,
			READ:= TRUE,
			TMOUT:= T#200ms,
			BUSY=> ,
			ERR=> ,
			ERRID=> );
		IF NOT fbAdsRead.BUSY THEN
			fbAdsRead( READ := FALSE );
			IF fbAdsRead.ERR THEN
				bErr := TRUE;
				nErrId := fbAdsRead.ERRID;
				nState := 16#999;
			ELSE
				nState := 16#20;
			END_IF
		END_IF

16#20: (* clear old interpolation Group *)

	fbClearGrp(
		bExecute:= TRUE,
		nGroupId:= nGroup,
		tTimeOut:= T#200ms);

	IF NOT fbClearGrp.bBusy THEN
		fbClearGrp(bExecute:= FALSE);
		IF NOT fbClearGrp.bErr THEN
			nState	:= 16#30;
		ELSE
			(* an error occured *)
			bErr		:= TRUE;
			nErrId	:= fbClearGrp.nErrId;
			nState	:= 16#999;
		END_IF
	END_IF


16#30: (* end *)
	bBusy := FALSE;
	nState := 0;


16#999:	(* Error *)
		bBusy := FALSE;
		nState := 0;
END_CASE

END_FUNCTION_BLOCK

// ---- POUs/Programy/PRG_Zaklejarka.TcPOU
PROGRAM PRG_Zaklejarka
VAR
	
	falownik3: FB_MX2;

	IFZaklejarka_FQ: INT;
	bFZaklejarka_CW: BOOL;
	bFZaklejarka_CCW: BOOL;
	bFZaklejarka_Reset: BOOL;
	krok				:INT;
	czas                 : ARRAY [0..100] OF TON ;
	b_Start AT %I* :BOOL;
	b_Stop AT %I* :BOOL;
		

	start: BOOL;
	bJog_F: BOOL;
	bJog_B: BOOL;
END_VAR

A_Falownik();
A_Automat_Zaklejarka();
	
		//IF GVL_HMI.bManual=TRUE THEN  ///TO NIE MOJE

IF GVL_HMI.bAuto=FALSE 	AND GVL_GLOBAL.tasmy_zaklejarka_cewka=TRUE	THEN		/// TO MOJE
bFZaklejarka_CCW:=TRUE;							
bFZaklejarka_CW:=0;
IFZaklejarka_FQ:=2000;

ELSIF GVL_HMI.bAuto=FALSE AND GVL_GLOBAL.tasmy_zaklejarka_cewka=FALSE THEN
	bFZaklejarka_CCW:=0;											
	bFZaklejarka_CW:=0;
(*ELSE

bFZaklejarka_CCW:=GVL_GLOBAL.bFZaklejarka_CCW;
bFZaklejarka_CW:=0;
*)
END_IF

ACTION A_Automat_Zaklejarka:
CASE Krok OF
	

	0:
			//IFZaklejarka_FQ:=2000;
		bFZaklejarka_CCW:=FALSE; 
	 IF start=TRUE AND GVL_HMI.bEnableZaklejarka=TRUE  THEN
		 
		 
		 Krok:=5;
		 
	 END_IF
	
	
	5:
		IFZaklejarka_FQ:=3000;
		bFZaklejarka_CCW:=TRUE; 
		GVL_GLOBAL.zamykacz_zaklejarka_auto:=FALSE;	
	
	IF	czas[1].Q=TRUE THEN
		
		Krok:=7;
	
	
	END_IF
	
	7:
	IF	GVL_Zak_IO.b_Czujnik_Karton=FALSE THEN /// tutaj można dodać że jak przez 30s nie przyjedzie karton to stop
		
	
	Krok:=10; 
	
	END_IF

	10:

	IF czas[2].Q=TRUE THEN 
	GVL_GLOBAL.zamykacz_zaklejarka_auto:=TRUE;	
	Krok:=15 ;
	END_IF 
	
	
	15:
	
	
	IF czas[0].Q=TRUE THEN 
	
	Krok:=20; 
		
	END_IF
	
	20:
	
	
	Krok:=5 ;
	
	
	

END_CASE
czas[1](IN:=GVL_Zak_IO.b_Czujnik_Karton, PT:=T#200MS);
czas[0](IN:=krok=15 , PT:=T#2S);
czas[2](IN:=krok=10 , PT:=T#500MS);

IF GVL_HMI.A_Start=TRUE AND GVL_HMI.bEnableZaklejarka=TRUE THEN 
start:=TRUE;
END_IF
			IF GVL_HMI.A_Stop=TRUE	OR GVL_HMI.bEnableZaklejarka=FALSE THEN
			start:=FALSE;	
			Krok:=0;
			bFZaklejarka_CCW:=FALSE; 
			
			END_IF
END_ACTION

ACTION A_Falownik:
falownik3
	(w_Status:=GVL_Omron.wOmron_Za_Status,
	ui_CzestotliwoscI:=IFZaklejarka_FQ,
	b_CCW:=bFZaklejarka_CW, 
	b_CW:=bFZaklejarka_CCW,
	b_Reset:=bFZaklejarka_Reset,
	w_ControlW=>GVL_Omron.wOmron_Za_Control,
 	ui_CzestotliwoscO=>GVL_Omron.iOmron_Za_SeVelo,);
END_ACTION

ACTION ACT_AutomaticMode:

END_ACTION

ACTION ACT_ManualMode:

END_ACTION

END_PROGRAM

// ---- POUs/Programy/PRG_Kartoniarka.TcPOU
PROGRAM PRG_Kartoniarka
VAR
		bTest2				:BOOL:=TRUE;
		falownik2			:FB_MX2;
		Falownik1			:FB_MX2;
		fb_Mag_POS			:FB_MX2_POS;
		F1_CW				:BOOL;
		F1_CCW				:BOOL;
		F1_FQ				:INT;
		L_Kolejny 			:INT;
		MagDocisk1			:BOOL;
		P_FIRST_CYCLE  		:R_TRIG;
		R_Pobranie_Kierwonica:R_TRIG;

		tm_error:  TIME := T#5S;
		errorTimer  :ARRAY[0..240] OF TON;
		Errors :ARRAY[0..100] OF BOOL;
		i_spr_blad : INT;
		Error_ind: bool;
	//balluff funkcja do zmiany I/o
	
	bSelect :BOOL;
	iIO_Link_Port :INT;
	iIndex :INT;
	iSubindex :INT;
	iDataLenght :UINT;
	arWrite_Data :ARRAY [0..20] OF BYTE;
	bStart :BOOL;
	arRead_Data :ARRAY[0..240] OF BYTE;
	bError :BOOL;
	
	//bloki do serwa
	S_Power :MC_Power;
	S_Move :MC_MoveAbsolute;
	S_Jog :MC_Jog;
	S_Reset :mc_reset;
	cz  :ARRAY[0..240] OF TON;
	czas  :ARRAY[0..240] OF TON;
	
	
	bEnable: BOOL;
	bJog_F: BOOL;
	bJog_B: BOOL;
	J_Vel: LREAL;
	bExecute: BOOL;
	Position: LREAL;
	Predkosc: LREAL;
	Automat: FB_K_Auto;
	F_Reset: BOOL;
	A_Error: BOOL;
	A_Error_ID: UDINT;
	Reset: BOOL;
	F2_CW: BOOL;
	F2_CCW: BOOL;
	F2_FQ: INT;
	Cz_M_D: INT;
	podjazd: BOOL;
	b_Stop_Kartoniarka: BOOL;
	
	bExecute_Mag: BOOL;
	bJogMinus_Mag: BOOL;
	bStop_Mag: BOOL;
	lrPosition_Mag: LREAL;
	lrVelocity_Mag: LREAL;
	lrAcc_Mag: LREAL;
	lrDcc_Mag: LREAL;
	bKoniecKartonow: BOOL;
	fbMagazyn: FB_Magazyn;
	bMagazynLaduj: BOOL;
	bMagazynDocisk: BOOL;
	bMagazynAutomat: BOOL;
	bResetMagazyn: BOOL;
	bMagazynZaladuj: BOOL;
	bMagazynZaladowany: BOOL;
	iMagazynPredkoscAuto: INT;
	bMagazynPodjazdAuto: BOOL;
	bMagazynCofniAuto: BOOL;
	abMagazynBlad: ARRAY [0..100] OF BOOL;
	MagAutomat: BOOL;
	bMagazynPodjazdManual: BOOL;
	bMagazynCofniManual: BOOL;
	
	fale: INT;
	MagDocisk: INT;
	K_Magazyn: FB_Magazyn;
END_VAR

VAR_INPUT
	bJogPlus_Mag: BOOL;
END_VAR

//automat
M_Automat();
//falowniki kartoniarka
M_F_Kartoniarka();
//serwa kartoniarka obsługa
M_K_Serwo();
//obsługa io-linka 
M_K_IO_Link();
//obsluga auto manual magazyn
A_FmagazynDocisk();
//obsługa przycisków kartoniarki
A_Przyciski_Kartoniarka();
//
A_Magazyn();
//A_Obsluga_bledow(); /// dodane moje
//obsługa manual auto 

	//IF GVL_HMI.bManual=TRUE THEN
IF GVL_HMI.bAuto=FALSE THEN			
	J_Vel:=100;
	bJog_F:=GVL_HMI.bHmiJogKF;
	bJog_B:=GVL_HMI.bHmiJogKB;	

END_IF

ACTION A_FmagazynDocisk:


	
	IF GVL_HMI.zaladowalem=TRUE AND  GVL_IO.Cz_M_D=FALSE AND gvl_hmi.bAuto=TRUE AND GVL_HMI.zaladuj=FALSE AND czas[0].Q=FALSE THEN
	
		iMagazynPredkoscAuto:=2000;
		bMagazynPodjazdAuto:=TRUE;
		GVL_HMI.zaladowalem:=TRUE;
		
	END_IF
	IF gvl_hmi.bAuto=TRUE  AND czas[2].Q=TRUE AND GVL_HMI.zaladuj=FALSE THEN
		

		iMagazynPredkoscAuto:=0;
		bMagazynPodjazdAuto:=FALSE;
	
	
	END_IF
		
	IF GVL_HMI.zaladuj=TRUE AND czas[1].Q=FALSE AND gvl_hmi.bAuto=TRUE THEN
		
		GVL_HMI.zaladowalem:=FALSE;
		iMagazynPredkoscAuto:=2000;
		bMagazynCofniAuto:=TRUE;
	END_IF
	IF czas[1].Q=TRUE THEN
		
		//iMagazynPredkoscAuto:=0;
		bMagazynCofniAuto:=FALSE;
		GVL_HMI.zaladuj:=FALSE; 
	
	END_IF
	
	czas[0](IN:=bMagazynPodjazdAuto=TRUE,PT:=T#10S);
	czas[1](IN:=bMagazynCofniAuto=TRUE,PT:=T#3S);
	czas[2](IN:=GVL_IO.Cz_M_D=TRUE,PT:=T#1S);
END_ACTION

ACTION A_Magazyn:
K_Magazyn(
	xPodjedz:=gvl_io.bStart, 
	xWydajKarton:=, 
	xKartonPobrany:=, 
	xCzPodjazd:=, 
	xCzTrzymacz1:=, 
	xCzTrzymacz2:=GVL_IO.bCzujnik_Trzymacz1, 
	xSilPodpych=>GVL_IO.K1K4, 
	xSilTrzymacz1=>GVL_IO.K1K1, 
	xSilTrzymacz2=>GVL_IO.K1K3, 
	xWydalemKarton=>, 
	xBlad=> );
END_ACTION

ACTION A_Obsluga_bledow:


// WYŚWIERLANIE NUMERU BŁĘDU 

FOR i_spr_blad:=0 TO 10 DO
	IF Errors[i_spr_blad]=TRUE THEN
		i_spr_blad:=GVL_HMI.INT_idError;
		Error_ind:=TRUE;
	END_IF
END_FOR

IF GVL_HMI.bReset=TRUE THEN
	Error_ind:=FALSE;
END_IF
END_ACTION

ACTION A_Przyciski_Kartoniarka:
IF  (gvl_hmi.A_Start=TRUE  OR  P_FIRST_CYCLE.Q=TRUE ) THEN GVL_IO.K1K5:=FALSE; GVL_IO.K1K7:=TRUE; L_Kolejny:=L_Kolejny+1; END_IF
IF gvl_hmi.A_Stop=TRUE THEN GVL_IO.K1K5:=TRUE; GVL_IO.K1K7:=FALSE;  END_IF
GVL_HMI.A_Start:=gvl_Io.b1K1;
GVL_HMI.A_Stop:=GVL_IO.b1K3;


P_FIRST_CYCLE(CLK:=GVL_HMI.Bit_Startu);
END_ACTION

ACTION M_Automat:
//Automat kartoniarka

Automat(
	Zasilanie:= GVL_HMI.bEnableKartoniarka,
	Start:= GVL_HMI.A_Start, 
	Stop:=GVL_HMI.A_Stop, 
	Reset:=GVL_GLOBAL.Error_reset_kart,
	kolejny:=GVL_HMI.Nastepny_Karton,
	Pauza:= , 
	Safety1:=GVL_SafetyFrom_RT2.bSAFETY_PermissionSS1,
	Safety2:=GVL_SafetyFrom_RT2.bSAFETY_PermissionSS2,
	W_Wys:= GVL_IO.Wyp_wys, 
	W_Cof:= GVL_IO.Wyp_cof, 
	Docisk_Wys:= GVL_IO.Skos_wyp, 
	Docisk_Cof:= GVL_IO.Skos_cof, 
	K1_Wys:= GVL_IO.Kl_1_wyp, 
	K1_Cof:= GVL_IO.Kl_1_cof, 
	K2_Wys:= GVL_IO.Kl_2_wyp, 
	K2_Cof:= GVL_IO.Kl_2_cof, 
	K_Dluga_Wyp:=GVL_IO.Zeb_Wyp , 
	K_Dluga_Cof:= GVL_IO.Zeb_Cof, 
	S_Ready:=S_Power.Active, 
	S_Run:= S_Move.Busy, 
	S_Done:=S_Move.Done,
	xKartonWydany:=K_Magazyn.xWydalemKarton,
	Pred_zad_podjazd:=GVL_Recipe.Predk_mag_pobranie,
	Pred_zad_odjazd:=GVL_Recipe.Predk_mag_odlozenie,
	S_KL_Dl=>GVL_GLOBAL.S_KL_Dl , 
	S_KL1_K=> GVL_global.S_KL1_K, 
	S_KL2_K=> GVL_global.S_KL2_K, 
	S_Wy=> GVL_global.S_Wy, 
	S_EXE=> bExecute, 
	S_Docisk=>GVL_GLOBAL.S_skos,
	F2_Run=>GVL_GLOBAL.F1_CW , //tutaj bylo samo F1_CW
	Pomp_V=>GVL_global.zaw_ssawki_auto, 
	Pozycja=>Position , 
	Predkosc=>Predkosc , 
	F2_CZ=>F1_FQ,
	Error_ind=>GVL_GLOBAL.Error_ind_kart,
	Error_numb=>GVL_GLOBAL.Error_numb_kart,
	xKartonZabrany=>K_Magazyn.xKartonPobrany,
	xWydajKarton=>K_Magazyn.xWydajKarton,
    );
END_ACTION

ACTION M_F_Kartoniarka:
//obsługa falownika taśm wyjazdowych 
	falownik2
	(w_Status:=GVL_Omron.wOmron_1_Status,
	ui_CzestotliwoscI:=F1_FQ,
	b_CCW:=F1_CW, // tutaj było samo F1_CW
	b_CW:=F1_CCW, // tutaj bylo F1_CCW
	b_Reset:=F_Reset,
			
	w_ControlW=>GVL_Omron.wOmron_1_Control,
 	ui_CzestotliwoscO=>GVL_Omron.iOmron_1_SeVelo,);
	
	

//-------------------------------obsługa AUTOMAT/MANUAL--------------------------------------------:

(*IF MagAutomat=TRUE THEN 
	
	F2_FQ:=iMagazynPredkoscAuto;
	F2_CW:=bMagazynPodjazdAuto;;
	F2_CCW:=bMagazynCofniAuto;
	
	
	
ELSIF MagAutomat=FALSE AND  GVL_AXIS.EC_Magazyn.NcToPlc.ActPos>5200 AND GVL_AXIS.EC_Magazyn.NcToPlc.ActPos<4300 THEN 
	

	F2_FQ:=1000;
	F2_CW:=bMagazynPodjazdManual;
	F2_CCW:=bMagazynCofniManual;
	*)
	IF GVL_HMI.bAuto=FALSE THEN 
		
	F2_FQ:=2000;
	F2_CW:=GVL_HMI.bHmiMagCw;
	F2_CCW:=GVL_HMI.bHmiMagCcw;
	
	ELSIF GVL_HMI.bAuto=TRUE THEN 
		
	F2_FQ:=iMagazynPredkoscAuto;
	F2_CW:=bMagazynCofniAuto;
	F2_CCW:=bMagazynPodjazdAuto;
	
	END_IF

//END_IF
IF GVL_HMI.bAuto=FALSE AND GVL_GLOBAL.falownik_pasow_cewka=TRUE THEN //moje 
	J_Vel:=100;
	F1_CW:=TRUE;
	F1_CCW:=0;
	F1_FQ:=2000; 
	
	ELSIF GVL_HMI.bAuto=FALSE AND GVL_GLOBAL.falownik_pasow_cewka=FALSE THEN
	J_Vel:=100;
	F1_CW:=0;
	F1_CCW:=0;
	F1_FQ:=0;
	
	ELSE
		J_Vel:=100;
		F1_CW:=GVL_GLOBAL.F1_CW;
		F1_CCW:=GVL_GLOBAL.F1_CCW;
	END_IF 
	

(*nie działa blok do osi
fb_Mag_POS(
	Ax:=GVL_AXIS.F_Magazyn , 
	Enc:=GVL_AXIS.EC_Magazyn.NcToPlc.ActPos , 
	ExecuteEn:=bExecute_Mag , 
	//En1:= , 
	JogPlus:=bJogPlus_Mag , 
	JogMinus:=bJogMinus_Mag , 
	Stop_Ex:=bStop_Mag , 
	Position:=lrPosition_Mag , 
	Velocity:=lrVelocity_Mag , 
	ACC:=lrAcc_Mag , 
	DCC:=lrDcc_Mag , 
	A_PosMx2=> , 
	A_V=> , 
	Error=> , 
	bDonePos=> , 
	Prawo=>,
	Lewo=> 
);

*)
END_ACTION

ACTION M_K_IO_Link:



	
		//załączenie kanałów io-link
		
		GVL_IO.IOLinkCh1T:=TRUE;
		
	

	
	//IO Link power
	
	gvl_IO.IOLinkCh1T:=TRUE;
END_ACTION

ACTION M_K_Serwo:
	
	//obsługa serwa
	
s_power(
	Axis:=GVL_AXIS.stAxis1 , 
	Enable:=GVL_AXIS.bEnable , 
	Enable_Positive:=GVL_AXIS.bEnable , 
	Enable_Negative:=GVL_AXIS.bEnable , 
	Override:=100.0 , 
	BufferMode:= , 
	Options:= , 
	Status=> , 
	Busy=> , 
	Active=> , 
	Error=> , 
	ErrorID=> );
	
	S_Reset(
	Axis:= GVL_AXIS.stAxis1, 
	Execute:=GVL_HMI.A_Stop , 
	Done=> , 
	Busy=> , 
	Error=> , 
	ErrorID=> );
		
	S_Jog(
	Axis:= GVL_AXIS.stAxis1, 
	JogForward:= bJog_B , 
	JogBackwards:=bJog_F , 
	Mode:= , 
	Position:= , 
	Velocity:= GVL_HMI.J_VelK, 
	Acceleration:= , 
	Deceleration:= , 
	Jerk:= , 
	Done=> , 
	Busy=> , 
	Active=> , 
	CommandAborted=> , 
	Error=> , 
	ErrorID=> );
	
	S_Move(
	Axis:=GVL_AXIS.stAxis1 , 
	Execute:= bExecute, 
	Position:=Position , 
	Velocity:=Predkosc , 
	Acceleration:= , 
	Deceleration:= , 
	Jerk:= , 
	BufferMode:= , 
	Options:= , 
	Done=> , 
	Busy=> , 
	Active=> , 
	CommandAborted=> , 
	Error=>A_Error , 
	ErrorID=>A_Error_ID
 );
END_ACTION

END_PROGRAM

// ---- POUs/FB/FB_MX2_POS.TcPOU
FUNCTION_BLOCK FB_MX2_POS
VAR
				
			FB_SetPos 				:MC_SetPosition;
			
			FB_MoveAbs				:MC_MoveAbsolute;
			FB_Jog					:MC_Jog;
			FB_McStop				:MC_Stop;
			Done					:BOOL;
			Busy					:BOOL;
			Er						:ARRAY[0..100] OF BOOL;
			A_Pos					:LREAL;
	fbMc_Power: MC_Power;
END_VAR

VAR_IN_OUT
	Ax								: AXIS_REF;
END_VAR

VAR_INPUT
	Enc								: LREAL;
	ExecuteEn						: BOOL;
	En1								: BOOL;
	JogPlus							: BOOL;
	JogMinus						: BOOL;
	Stop_Ex							: BOOL;
	Position						: LREAL;
	Velocity						: LREAL;
	ACC								: LREAL;
	DCC								: LREAL;
END_VAR

VAR_OUTPUT
	A_PosMx2						: LREAL;
	A_V								: LREAL;
	Error							: BOOL;
	bDonePos						: BOOL;
	Prawo							: BOOL;
	Lewo							: BOOL;	
END_VAR

IF JogPlus=FALSE AND JogMinus=FALSE  THEN //AND Busy=FALSE
	

FB_SetPos(
	Axis:=AX , 
	Execute:=TRUE , 
	Position:=Enc , 
	Mode:= , 
	Options:= , 
	Done=> , 
	Busy=> , 
	Error=>Er[0] , 
	ErrorID=> );
	
	
FB_SetPos(
	Axis:=AX , 
	Execute:=FALSE , 
	Position:=Enc , 
	Mode:= , 
	Options:= , 
	Done=> , 
	Busy=> , 
	Error=>Er[1] , 
	ErrorID=> );
END_IF

FB_Jog(
	Axis:=AX , 
	JogForward:=JogPlus , 
	JogBackwards:=JogMinus , 
	Mode:=MC_JOGMODE_CONTINOUS , 
	Position:= , 
	Velocity:=Velocity , 
	Acceleration:=ACC , 
	Deceleration:=DCC , 
	Jerk:= , 
	Done=> , 
	Busy=> , 
	Active=> , 
	CommandAborted=> , 
	Error=>Er[2] , 
	ErrorID=> );
	
	
FB_MoveAbs(
	Axis:=AX , 
	Execute:=ExecuteEn , 
	Position:=Position , 
	Velocity:=Velocity , 
	Acceleration:=ACC , 
	Deceleration:=DCC , 
	Jerk:= , 
	BufferMode:=MC_Aborting , 
	Options:= , 
	Done=> , 
	Busy=>Busy , 
	Active=> , 
	CommandAborted=> , 
	Error=>Er[3] , 
	ErrorID=> );	
	
FB_McStop(
	Axis:=AX , 
	Execute:=Stop_Ex , 
	Deceleration:=DCC , 
	Jerk:= , 
	Options:= , 
	Done=> , 
	Busy=> , 
	Active=> , 
	CommandAborted=> , 
	Error=> Er[4], 
	ErrorID=> );
	
	A_PosMx2:=Ax.NcToPlc.ActPos;
		
	Error:=Er[0]=TRUE OR Er[1]=TRUE OR Er[2]=TRUE OR Er[3]=TRUE OR Er[4]=TRUE;
	
	
	IF  Ax.NcToPlc.ActVelo<700.0 AND   Ax.NcToPlc.ActVelo>0 AND Ax.NcToPlc.ActVelo <>0.0 THEN
		
		
	A_V:=700;
	LEWO:=FALSE;
	PRAWO:=TRUE;
	ELSIF Ax.NcToPlc.ActVelo>700.0 AND   Ax.NcToPlc.ActVelo>0 AND Ax.NcToPlc.ActVelo <>0.0 THEN
		
	A_V:=Ax.NcToPlc.ActVelo;
	LEWO:=FALSE;
	PRAWO:=TRUE;
	
	ELSIF Ax.NcToPlc.ActVelo =0 THEN
		
		LEWO:=FALSE;
		PRAWO:=FALSE;
	
	END_IF
	
	IF  Ax.NcToPlc.ActVelo>-700.0 AND   Ax.NcToPlc.ActVelo<0 AND Ax.NcToPlc.ActVelo <>0.0 THEN
		
		
	A_V:=700;
	LEWO:=TRUE;
	PRAWO:=FALSE;
	ELSIF Ax.NcToPlc.ActVelo<-700.0 AND Ax.NcToPlc.ActVelo <>0.0 THEN
		
	A_V:=Ax.NcToPlc.ActVelo;
	LEWO:=TRUE;
	PRAWO:=FALSE;
	
	ELSIF Ax.NcToPlc.ActVelo =0 THEN
		
		LEWO:=FALSE;
		PRAWO:=FALSE;
	
	END_IF
	

	
	IF Ax.NcToPlc.ActPos<Position+10.0 AND Ax.NcToPlc.ActPos>Position-10.0 THEN
	bDonePos:=TRUE;
ELSE
	bDonePos:=FALSE;	
END_IF;

fbMc_Power(
	Axis:=AX , 
	Enable:=TRUE , 
	Enable_Positive:=TRUE , 
	Enable_Negative:=TRUE , 
	Override:= , 
	BufferMode:= , 
	Options:= , 
	Status=> , 
	Busy=> , 
	Active=> , 
	Error=> , 
	ErrorID=> );

END_FUNCTION_BLOCK

// ---- POUs/FB/FB_K_Auto.TcPOU
FUNCTION_BLOCK FB_K_Auto
VAR_INPUT
	Zasilanie:bool;
	Start:BOOL;
	Stop:BOOL;
	Pauza:BOOL;
	W_Wys:BOOL;
	W_Cof:BOOL;
	Docisk_Wys:BOOL;
	Docisk_Cof:BOOL;
	K1_Wys:BOOL;
	K1_Cof:BOOL;
	K2_Wys:BOOL;
	K2_Cof:BOOL;
	K_Dluga_Wyp:BOOL;
	K_Dluga_Cof:BOOL;
	S_Ready:BOOL;
	S_Run:BOOL;
	S_Done:BOOL;
	kolejny: BOOL;
	Safety1 : BOOL;
	Safety2  : BOOL;
	Pred_zad_podjazd: LREAL;
	Pred_zad_odjazd: LREAL;
	Reset: BOOL;
	xKartonWydany :BOOL;
	
END_VAR
VAR_OUTPUT
	S_KL_Dl:BOOL;
	S_KL1_K:BOOL;
	S_KL2_K:BOOL;
	S_Wy:BOOL;
	S_EXE:BOOL;	
	S_Docisk:BOOL;
	F2_Run:BOOL;	
	Pomp_V:BOOL;
	Pozycja:LREAL;
	Predkosc:LREAL;
	F2_CZ:INT;
	Error_ind: BOOL;
	Error_numb: INT;
	xKartonZabrany:BOOL;
	xWydajKarton:BOOL;
	
	
END_VAR
VAR
	Seq :INT;
	Czas :ARRAY[0..100] OF TON;
	CZ :TON;
	przeliczenie :INT;
	alarm_int : INT:=3;
	
END_VAR

CASE seq OF
	

0:(**)
	S_KL_Dl:=FALSE;
	S_KL1_K:=FALSE;
	S_KL2_K:=FALSE;
	S_Wy:=FALSE;
	S_EXE:=FALSE;
	S_Docisk:=FALSE;
	F2_Run:=FALSE;
	Pomp_V:=FALSE;
	F2_CZ:=0;
	
	xKartonZabrany:=FALSE;

	IF start=TRUE AND Safety1=TRUE AND Safety2=TRUE AND Zasilanie=TRUE THEN
		
	Seq:=5;

	END_IF
	

4:(*start kolejnego cyklu *)

	
	S_KL_Dl:=FALSE;
	S_KL1_K:=FALSE;
	S_KL2_K:=FALSE;
	S_Wy:=FALSE;
	S_EXE:=FALSE;
	S_Docisk:=FALSE;
	//F2_Run:=FALSE;
	Pomp_V:=FALSE;
	//F2_CZ:=0;
	
	IF kolejny=TRUE THEN
		
	Seq:=5;

	END_IF

5:(**)
	
	IF W_Cof=TRUE AND Docisk_Cof=TRUE AND K1_Cof=TRUE AND K2_Cof=TRUE AND K_Dluga_Cof=TRUE AND S_Ready=TRUE  THEN
		
	F2_CZ:=2000;
	F2_Run:=TRUE;

	Seq:=10;
	END_IF


10:(**)
	Predkosc:=Pred_zad_podjazd;		/// 900
	Pozycja:=600;
	
	IF S_Ready=TRUE THEN
	
		S_EXE:=TRUE;
	
	END_IF
	
	IF S_Run=TRUE THEN
		S_EXE:=FALSE;
		Seq:=15;
	
	END_IF

15:(**)
	IF S_Done=TRUE THEN
		Pomp_V:=TRUE;    // czy został zamontowany czujnik podcisnienie???
		xWydajKarton:=TRUE;
		
		Seq:=17; 
	END_IF
17:(**)	
		//IF GVL_IO.Vacuostat=TRUE THEN
	//	IF Czas[11].q=TRUE THEN 
		Seq:=20; 
		//END_IF
		//END_IF



20:(**)
	Pozycja:=225-((GVL_Recipe.szer_kartonu)/2);//dla malego kartonu bylo 156 //dla kartonu 370x370 was 40 
	Predkosc:=Pred_zad_odjazd;
	IF czas[0].Q=TRUE AND S_Ready=TRUE AND xKartonWydany=TRUE THEN
		xWydajKarton:=FALSE;	
	 S_EXE:=TRUE;
	 
	
	END_IF

	IF S_Run=TRUE THEN 

	Seq:=25;
	
	END_IF

25:(**)
	IF S_Done=TRUE THEN
		S_EXE:=FALSE;
		S_Docisk:=TRUE;
		xKartonZabrany:=TRUE;
		seq:=30;
	
	END_IF

30:(**)
	
	IF 	Docisk_Wys=TRUE THEN 
		xKartonZabrany:=FALSE;
	S_KL1_K:=TRUE;
	S_KL2_K:=TRUE;
		seq:=35;
	END_IF
	

35:(**)
	IF K1_Wys=TRUE AND K2_Wys=TRUE THEN
		S_KL_Dl:=TRUE;
		
		seq:=40;
	END_IF
40:(**)

	IF K_Dluga_Wyp=TRUE AND Czas[1].Q=TRUE THEN
		Pomp_V:=FALSE;
		seq:=42;
	END_IF
	
42:
	Pozycja:=225-((GVL_Recipe.szer_kartonu)/2)-20;//dla malego kartonu bylo 156 //dla kartonu 370x370 was 40
	Predkosc:=800; /// predkosc odjazdu do home
	IF  S_Ready=TRUE AND S_Run=FALSE THEN
		
	 S_EXE:=TRUE;
	 
	
	END_IF

	IF S_Run=TRUE THEN 
		
	Seq:=44;
	
	END_IF
44:
	IF S_Done=TRUE THEN
		S_Wy:=TRUE;
		Seq:=45;
	END_IF
	

45:(**)
	IF W_Wys=TRUE AND Czas[2].Q=TRUE  THEN
		
		S_KL_Dl:=FALSE;
		S_KL1_K:=FALSE;
		S_KL2_K:=FALSE;
		S_Wy:=FALSE;
		
		
		seq:=50;
	END_IF

50:(**)
	IF  W_Cof=TRUE  AND K1_Cof=TRUE AND K2_Cof=TRUE AND K_Dluga_Cof=TRUE THEN
		
	S_Docisk:=FALSE;
	seq:=4;
	END_IF

1000:(**)// Errors
	
	Error_ind:=TRUE;
	F2_Run:=FALSE;
	Pomp_V:=FALSE;  
	IF Reset=TRUE THEN
		Error_ind:=FALSE;
		Error_numb:=0;
		alarm_int:=3;
		seq:=0;
	END_IF

END_CASE

Czas[0](IN:=seq=20, PT:=T#450MS);
Czas[1](IN:=seq=40, PT:=T#0.5S);
Czas[2](IN:=seq=45, PT:=T#0.5S);

//czasowki do bledow
Czas[3](IN:=seq=5, PT:=T#5S); //Błąd gotowości do pracy
//Czas[4](IN:=seq=15, PT:=T#5S);
Czas[5](IN:=seq=25, PT:=T#5S); // Nie osiągnięto pozycji składania kartonu
Czas[6](IN:=seq=30, PT:=T#5S); // Docisk się nie wysunął
Czas[7](IN:=seq=35, PT:=T#5S); // Błąd klap
Czas[8](IN:=seq=40, PT:=T#5S); // Błąd wypychacz
Czas[9](IN:=seq=44, PT:=T#5S); // Błąd pozycji oczekiwania
Czas[10](IN:=seq=50, PT:=T#5S); // Błąd kończenia cyklu... kartoniarka nie przechodzi do stanu początkowego
Czas[11](IN:=GVL_IO.K1K3=TRUE, PT:=T#1S); // Błąd kończenia cyklu... kartoniarka nie przechodzi do stanu początkowego
// Obsługa błędów

IF Reset= FALSE THEN
FOR alarm_int:=3 TO 10 DO 
IF Czas[alarm_int].Q=TRUE THEN
	Error_numb:=alarm_int+100; // DLA KART. +100 DLA ZAKLEJARKI +200 ITD
	seq:=1000;
END_IF	
END_FOR
END_IF

IF stop=TRUE OR Safety1=FALSE OR Safety2=FALSE OR Zasilanie=FALSE  THEN 
	
	seq:=0;
		F2_Run:=FALSE;
		

	

END_IF

END_FUNCTION_BLOCK

// ---- POUs/FB/FB_Magazyn.TcPOU
FUNCTION_BLOCK FB_Magazyn
VAR_INPUT
	xPodjedz :BOOL;
	xWydajKarton :BOOL;
	xKartonPobrany :BOOL;
	xCzPodjazd :BOOL;
	xCzTrzymacz1 :BOOL;
	xCzTrzymacz2 :BOOL;
	bStop 		:BOOL;
	
END_VAR
VAR_OUTPUT
	xSilPodpych :BOOL;
	xSilTrzymacz1 :BOOL;
	xSilTrzymacz2 :BOOL;
	xWydalemKarton :BOOL;
	xBlad					:ARRAY[0..100]  OF BOOL;
	
END_VAR

VAR
	czas					: ARRAY[0..100] OF TON;
	seq						: INT;
END_VAR

CASE seq OF 
	
0:(*inicjalizacja*)
	xSilPodpych:=FALSE;
	xSilTrzymacz1:=TRUE;
	xSilTrzymacz2:=FALSE;
	xWydalemKarton:=FALSE;	
	IF xPodjedz=TRUE THEN	
	seq:=5; 	
	END_IF
5:(*wlacza silownik podjazdu czeka sekunde *)

	xSilPodpych:=TRUE;
	xSilTrzymacz1:=TRUE;
	xSilTrzymacz2:=FALSE;
	IF czas[0].Q=TRUE THEN 
		seq:=10;
	END_IF
10:(*cofa silownik podjazdu *)
	xSilTrzymacz1:=FALSE;
	xSilTrzymacz2:=FALSE;
	IF xWydajKarton=TRUE THEN
		seq:=15;
	END_IF
15:(*opóźnienie popychu*)
IF czas[3].Q=TRUE THEN
	xSilPodpych:=FALSE;
	seq:=16;
END_IF
	
16:(*wydaje karton done zrobione *) 
	xSilPodpych:=FALSE;
	xSilTrzymacz1:=FALSE;
	xSilTrzymacz2:=TRUE;	
	IF xCzTrzymacz1=TRUE THEN
		xWydalemKarton:=TRUE;
		seq:=20;
	END_IF	
	
20:(*opoznienie trzymacza 2 *)
	
	xWydalemKarton:=FALSE;
	IF czas[1].Q=TRUE  AND xKartonPobrany=TRUE  THEN
	xSilTrzymacz1:=TRUE;
	xSilTrzymacz2:=FALSE;
	seq:=25;
	END_IF
25:(*popychacz z opóźnieniem*)
IF czas[2].Q=TRUE THEN
	xSilPodpych:=TRUE; 
	seq:=5;
END_IF


	
END_CASE
			czas[0](IN:=seq=5,PT:=T#3S);
			czas[1](IN:=seq=20,PT:=T#1S);
			czas[2](IN:=seq=25,PT:=T#1S);
			czas[3](IN:=seq=15,PT:=T#1S);
			
			//jak stop to zeruj seq
				
		IF bStop THEN	
			seq:=0;
		END_IF

END_FUNCTION_BLOCK

// ---- POUs/Programy/PRG_Kierownica.TcPOU
PROGRAM PRG_Kierownica
VAR
	

	F_Kierownica: FB_MX2;
	
	b_FK_CCW: BOOL;
	b_FK_CW: BOOL;
	b_FK_Reset: BOOL;
	
	//serwo 
	
	S_K_Power :MC_Power;
	S_K_Move :MC_MoveAbsolute;
	S_K_Jog :MC_Jog;
	S_K_Reset :mc_reset;
	fb_Home_Kierownica :MC_Home;
	
	bEnable: BOOL;
	bExecute: BOOL;
	Position: LREAL;
	Predkosc: LREAL;
	A_Error: BOOL;
	A_Error_ID: UDINT;
	bJog_F: BOOL;
	bJog_B: BOOL;
	J_Vel: LREAL;
	Reset: BOOL;
	ui_FKCzestotliwosc: INT;
	
	bHomeExe: BOOL;
	FB_Auto_Kierownica: FB_Kierownica;
	Pozycja_Kierownica: LREAL;
	bSDone: BOOL;
	bSBusy: BOOL;
	bReady: BOOL;
	
	//liczniki
	licznik1_rzedow: FB_Licznik;
	licznik2_rzedow: FB_Licznik;
	licznik3_rzedow: FB_Licznik;
	licznik4_rzedow: FB_Licznik;
	licznik5_rzedow: FB_Licznik;
	licznik_suma: INT; 
	// POMOCNICZE ZMIENNE
	ii : INT;
	TESTOWO: BOOL;
	predko: LREAL;
	pozycjaKier: LREAL;
	Error_ind: BOOL;
	Error_numb: INT;
	bStop: BOOL;
END_VAR

//falownik kierwonicy 
A_K_Falownik();
//serwo kierwoniczy 
A_Serwo();
A_Auto_Kierownica();
//A_Liczenie_butelek();

IF GVL_HMI.bAuto=FALSE THEN			
	J_Vel:=100;
	
	IF Pozycja_Kierownica>= 122 AND GVL_HMI.bHmiJogF=TRUE THEN
		bJog_F:=0;
		pozycjaKier:=122;
		ELSE
		bJog_F:=GVL_HMI.bHmiJogF;
	END_IF
		
	IF Pozycja_Kierownica<= -115 AND GVL_HMI.bHmiJogB=TRUE THEN
		bJog_B:=0;
		pozycjaKier:=-115;
		ELSE
		bJog_B:=GVL_HMI.bHmiJogB;
	END_IF
	
END_IF

ACTION A_Auto_Kierownica:
FB_Auto_Kierownica(
	b_czujnik_wejsciowy:=GVL_IO_K.b4B8 , 
	b_czujnik_K1:=GVL_IO_K.b4B1 , 
	b_czujnik_K2:=GVL_IO_K.b4B2 , 
	b_czujnik_K3:=GVL_IO_K.b4B3 , 
	b_czujnik_K4:=GVL_IO_K.b4B4 , 
	b_czujnik_K5:=GVL_IO_K.b4B5 , 
	b_Kon2:=GVL_IO_K.b4B6 , 
	b_Kon1:=GVL_IO_K.b4B7 ,
	Zasilanie:=GVL_HMI.bEnableKierownica,
	automat:= gvl_hmi.bAuto AND GVL_HMI.bEnableKierownica,
	b_Start:= , 
	b_Start1:= GVL_HMI.A_Start, 
	b_Stop:= GVL_HMI.A_Stop, 
	bS_Ready:=bReady , 
	bS_Run:=bSBusy , 
	bS_Done:=bSDone , 
	LR_Pozycja_Zadana:= , 
	b_Pobral:= GVL_GLOBAL.Ploter_pobral , 
	int_Licznik_zadana:=GVL_RECIPE.Il_rzedow, 
	int_Kieszen_zadana:=GVL_RECIPE.Il_kolumn , 
	LR_EPozycja=>pozycjaKier , 
	LR_Predkosc=> predko, 
	bS_Enable=> , //???
	bS_Exe=>bExecute , 
	b_Odbierz=> GVL_GLOBAL.Zabierz_Z_Kierownicy , // tutaj sygnał do pobrania oraz sprawdzenia stanu (ilosci butelek)
	b_Hamulec1=>GVL_IO_K.bK1, 
	b_Hamulec2=>GVL_IO_K.bK2, 
	Kier_CCw=>gvl_global.b_FK_CCW,
	Kier_Cw=>);
END_ACTION

ACTION A_K_Falownik:
F_Kierownica
	(w_Status:=GVL_Omron.wOmron_Kier_Status,
	ui_CzestotliwoscI:=ui_FKCzestotliwosc,
	b_CCW:=b_FK_CCW,
	b_CW:=b_FK_CW,
	b_Reset:=b_FK_Reset,
	w_ControlW=>GVL_Omron.wOmron_Kier_Control,
 	ui_CzestotliwoscO=>GVL_Omron.iOmron_Kier_SeVelo,);

//automat manual kierownica 
GVL_IO.Vacuostat;

	//IF GVL_HMI.bManual=TRUE THEN
IF GVL_HMI.bAuto=FALSE AND GVL_GLOBAL.falownik_podajnik_kier_cewka=TRUE AND GVL_HMI.bEnableKierownica=TRUE THEN
	Predkosc:=200;
	b_FK_CCW:=TRUE;
	b_FK_CW:=0;
	ui_FKCzestotliwosc:=1000;
ELSIF GVL_HMI.bAuto=FALSE OR GVL_IO.b1K3 THEN
		
	Predkosc:=0;
		b_FK_CCW:=FALSE;
		b_FK_CW:=FALSE;	
ELSIF GVL_HMI.bAuto=TRUE AND GVL_HMI.bEnableKierownica=TRUE THEN
		Predkosc:=200;
		predko:=200;
		ui_FKCzestotliwosc:=4000;
		b_FK_CCW:=GVL_GLOBAL.b_FK_CCW;
		b_FK_CW:=0;
END_IF
END_ACTION

ACTION A_Liczenie_butelek:
licznik1_rzedow(c_inkrement:=GVL_IO_K.b4B1,czas:=T#0.2S,c_stan=>GVL_GLOBAL.stan_licz[1]);
licznik2_rzedow(c_inkrement:=GVL_IO_K.b4B2,czas:=T#0.2S,c_stan=>GVL_GLOBAL.stan_licz[2]);
licznik3_rzedow(c_inkrement:=GVL_IO_K.b4B3,czas:=T#0.2S,c_stan=>GVL_GLOBAL.stan_licz[3]);
licznik4_rzedow(c_inkrement:=GVL_IO_K.b4B4,czas:=T#0.2S,c_stan=>GVL_GLOBAL.stan_licz[4]);
licznik5_rzedow(c_inkrement:=GVL_IO_K.b4B5,czas:=T#0.2S,c_stan=>GVL_GLOBAL.stan_licz[5]);


licznik_suma:=GVL_GLOBAL.stan_licz[1]+GVL_GLOBAL.stan_licz[2]+GVL_GLOBAL.stan_licz[3]+GVL_GLOBAL.stan_licz[4]+GVL_GLOBAL.stan_licz[5];

IF GVL_GLOBAL.Zabierz_Z_Kierownicy=TRUE  AND GVL_HMI.Wymus_pobranie=FALSE THEN 
		
 			IF GVL_Recipe.Il_kolumn*GVL_Recipe.Il_rzedow=licznik_suma THEN
			GVL_GLOBAL.reset_licznik:= TRUE;
			ELSE
			GVL_GLOBAL.Error_pakowaniA:=TRUE;
			GVL_GLOBAL.Error_numb_kier:=311; // 311 błąd liczenia kierownica
			GVL_GLOBAL.Zabierz_Z_Kierownicy:=FALSE; // Cofamy zgode na pobranie
			END_IF
			
END_IF

IF GVL_HMI.ErrorResetKier:=TRUE AND GVL_GLOBAL.Error_numb_kier=311 THEN 
	licznik_suma:=0;
	GVL_GLOBAL.Error_pakowania:=FALSE;
	GVL_GLOBAL.Error_numb_kier:=0;
END_IF

IF GVL_HMI.Wymus_pobranie=TRUE THEN
	GVL_GLOBAL.Zabierz_Z_Kierownicy:=TRUE;
	GVL_GLOBAL.reset_licznik:= TRUE;
END_IF
END_ACTION

ACTION A_Serwo:
	
	//obsługa serwa
	
S_K_Power(
	Axis:=GVL_AXIS.stAxis2 , 
	Enable:=GVL_AXIS.bEnable , 
	Enable_Positive:=GVL_AXIS.bEnable , 
	Enable_Negative:=GVL_AXIS.bEnable , 
	Override:=100.0 , 
	BufferMode:= , 
	Options:= , 
	Status=>bReady , 
	Busy=> , 
	Active=> , 
	Error=> , 
	ErrorID=> );
	
	S_K_Reset(
	Axis:= GVL_AXIS.stAxis2, 
	Execute:=GVL_HMI.ErrorResetKier , 
	Done=> , 
	Busy=> , 
	Error=> , 
	ErrorID=> );
		
	S_K_Jog(
	Axis:= GVL_AXIS.stAxis2, 
	JogForward:= bJog_F , 
	JogBackwards:=bJog_B , 
	Mode:= , 
	Position:= , 
	Velocity:= GVL_HMI.J_Vel, 
	Acceleration:= , 
	Deceleration:= , 
	Jerk:= , 
	Done=> , 
	Busy=> , 
	Active=> , 
	CommandAborted=> , 
	Error=> , 
	ErrorID=> );
	
	S_K_Move(
	Axis:=GVL_AXIS.stAxis2 , 
	Execute:= bExecute,//bExecute, 
	Position:=pozycjaKier ,//Position , 
	Velocity:=predko ,//Predkosc , 
	Acceleration:= , 
	Deceleration:= , 
	Jerk:= , 
	BufferMode:= , 
	Options:= , 
	Done=>bSDone , 
	Busy=>bSBusy , 
	Active=> , 
	CommandAborted=> , 
	Error=>A_Error , 
	ErrorID=>A_Error_ID);
 Pozycja_Kierownica:=GVL_AXIS.stAxis2.NcToPlc.ActPos;
 
 //home serwa 
 
 

	 fb_Home_Kierownica(
	Axis:= GVL_AXIS.stAxis2, 
	Execute:= bHomeExe, 
	Position:=0 , 
	HomingMode:=MC_Direct , 
	BufferMode:= , 
	Options:= , 
	bCalibrationCam:= , 
	Done=> , 
	Busy=> , 
	Active=> , 
	CommandAborted=> , 
	Error=> , 
	ErrorID=> );
END_ACTION

ACTION ACT_AutomaticMode:

END_ACTION

ACTION ACT_ManualMode:

END_ACTION

END_PROGRAM

// ---- POUs/FB/FB_Kierownica.TcPOU
FUNCTION_BLOCK FB_Kierownica
VAR_INPUT
	
			b_czujnik_wejsciowy 	:BOOL;
			b_czujnik_K1 			:BOOL;
			b_czujnik_K2 			:BOOL;
			b_czujnik_K3 			:BOOL;
			b_czujnik_K4 			:BOOL;
			b_czujnik_K5 			:BOOL;
			b_Kon2 					:BOOL;
			b_Kon1 					:BOOL;
			Zasilanie				:BOOL;
			b_Start					:BOOL;
			b_Start1				:BOOL;
			b_Stop					:BOOL;
			bS_Ready				:BOOL;
			bS_Run					:BOOL;
			bS_Done					:BOOL;
			LR_Pozycja_Zadana				:ARRAY[1..5] OF LREAL;
			b_Pobral 				:BOOL;
			int_Licznik_zadana      :INT;
			int_Kieszen_zadana 		:INT;
			automat					:BOOL;
END_VAR
VAR_OUTPUT
	
			LR_EPozycja				:LREAL;
			LR_Predkosc				:LREAL;
			bS_Enable				:BOOL;
			bS_Exe					:BOOL;
			b_Odbierz				:BOOL;
			b_Hamulec1 				:BOOL;
			b_Hamulec2 				:BOOL;
			Kier_CCW				:BOOL;
			Kier_CW					:BOOL;
END_VAR
VAR
	
			int_Kieszen				:INT :=1;
			int_Licznik				:INT; //liczenie ktora butelka w kasecie
			int_LicznikCheck		:ARRAY[1..5] OF INT; //liczenie ktora butelka w kasecie
			czas					:ARRAY[0..100] OF TON;
			Seq						:INT;
			Seq1						:INT;
			zaladowal				:BOOL;
	i: INT;
END_VAR

LR_Pozycja_Zadana[1]:=-115;	
LR_Pozycja_Zadana[2]:=-53;
LR_Pozycja_Zadana[3]:=7;
LR_Pozycja_Zadana[4]:=63;
LR_Pozycja_Zadana[5]:=122;


CASE seq OF
	

	0:
		//int_Kieszen:=1;
		
	IF (b_Start=TRUE OR b_Start1=TRUE)  AND bS_Ready=TRUE AND Zasilanie=TRUE  THEN
		b_Hamulec1:=TRUE;
		b_Hamulec2:=TRUE;
		
		IF bS_Ready=FALSE THEN 
			
			bS_Enable:=TRUE;
		END_IF
		
		
		IF bS_Ready=TRUE THEN
			seq:=5;
		END_IF
	
	
	END_IF
	
	
	5:
	
	
	
	LR_EPozycja:=LR_Pozycja_Zadana[int_Kieszen];
	LR_Predkosc:=350;
	b_Start:=FALSE;

	IF  b_Kon1=TRUE AND b_Kon2=TRUE THEN
	bS_Exe:=TRUE;
	END_IF
	
	IF bS_Run=TRUE THEN
	seq:=10;

	END_IF
	
	10:
	IF bS_Done=TRUE THEN
	bS_Exe:=FALSE;
	
	IF b_Odbierz=FALSE	THEN 
		b_Hamulec1:=FALSE;
		b_Hamulec2:=FALSE;
		
		END_IF
	seq:=0;
	
	END_IF
	


	
	
END_CASE
CASE seq1 OF
0:

			b_Start:=TRUE;
			seq1:=3;

3:
			//IF Czas[0].Q=FALSE THEN
				
			seq1:=5;
			
			//END_IF
			//int_Licznik	:=0;//zerowanie kieszeni 
			
			
5:

			IF Czas[0].Q=TRUE THEN
				
			seq1:=10;
			
			END_IF
			
10://inkremetnowanie licznika przejchala butelka 
			
			int_Licznik:=int_Licznik+1; 
			seq1:=15;
15:	
			IF int_Licznik=int_Licznik_zadana AND int_Kieszen<int_Kieszen_zadana+1 THEN
			int_Kieszen:=int_Kieszen+1;
			int_Licznik:=0;
			
			seq1:=25;	
			
			
			END_IF
		
	
			IF int_Kieszen=int_Kieszen_zadana+1 THEN
					
			GVL_GLOBAL.reset_licznik:=TRUE; ///moje
			
				b_Odbierz:=TRUE;
				int_Kieszen:=1;
				seq1:=25;	
			END_IF

			
			IF Czas[6].Q=TRUE THEN
			
						seq1:=3;
			
			END_IF
		
			

			
			
25:(*blokowanie silownika odblokowane dopiero jak przestawi sie kierownica na nastepną pozycję *)
		b_Hamulec1:=TRUE;
		b_Hamulec2:=TRUE;
		seq1:=30;	
			
30:(*startowanie serwa i czekanie jak pojedzie*)
		IF b_Kon2=TRUE AND b_Kon1=TRUE AND Czas[7].Q=TRUE THEN
			
		b_Start:=TRUE;
		seq1:=35;	
		END_IF

35:(*czekanie aż serwo wykona ruch jak wykona to skocz do 0:*)
		b_Start:=FALSE;
		
		IF bS_Done=TRUE  THEN
		seq1:=40;
		END_IF
40:(**)


		IF b_Odbierz=FALSE	THEN 
		b_Hamulec1:=FALSE;
		b_Hamulec2:=FALSE;
		seq1:=3;
		END_IF
END_CASE





Czas[0](IN:=b_czujnik_wejsciowy, PT:=T#20MS);
Czas[1](IN:=b_czujnik_K1, PT:=T#100MS);
Czas[2](IN:=b_czujnik_K2, PT:=T#100MS);
Czas[3](IN:=b_czujnik_K3, PT:=T#100MS);
Czas[4](IN:=b_czujnik_K4, PT:=T#100MS);
Czas[5](IN:=b_czujnik_K5, PT:=T#100MS);
Czas[6](IN:=b_czujnik_wejsciowy=FALSE, PT:=T#25MS);
Czas[7](IN:=seq1=30, PT:=T#500MS);
IF b_Stop=TRUE OR Zasilanie=FALSE OR automat=FALSE THEN
		
	seq:=0;
	Kier_CCW:=FALSE;
	Kier_CW:=FALSE;
	END_IF
IF b_Start1=TRUE AND Zasilanie=TRUE THEN	
	
	Kier_CCW:=TRUE;
	Kier_CW:=FALSE;
	END_IF
	IF b_pobral=TRUE THEN
		
	
	
	FOR i:=1 TO 5 BY 1 DO 
		
	int_LicznikCheck[i]:=0;
	END_FOR
 
	
	
	END_IF
	
	IF b_Pobral=TRUE THEN
			
			b_Odbierz:=FALSE;
					
			END_IF

END_FUNCTION_BLOCK

